LIN {X 0,Y 124.786,Z 596.16,A -85,B 0,C 180,E1 -33288.67,E2 -33288.67} C_VEL
LIN {X 0,Y 121.331,Z 587.817,A -85,B 0,C 180,E1 -33295.862,E2 -33295.862} C_VEL
LIN {X 0,Y 119.937,Z 579.475,A -85,B 0,C 180,E1 -33301.975,E2 -33301.975} C_VEL
LIN {X 0,Y 119.69,Z 571.877,A -85,B 0,C 180,E1 -33306.721,E2 -33306.721} C_VEL
LIN {X 0,Y 119.661,Z 563.812,A -85,B 0,C 180,E1 -33310.967,E2 -33310.967} C_VEL
LIN {X 0,Y 119.744,Z 553.937,A -85,B 0,C 180,E1 -33315.262,E2 -33315.262} C_VEL
LIN {X 0,Y 120.033,Z 541.878,A -85,B 0,C 180,E1 -33319.604,E2 -33319.604} C_VEL
LIN {X 0,Y 120.66,Z 528.353,A -85,B 0,C 180,E1 -33323.521,E2 -33323.521} C_VEL
LIN {X 0,Y 121.53,Z 514.293,A -85,B 0,C 180,E1 -33326.761,E2 -33326.761} C_VEL
LIN {X 0,Y 122.326,Z 501.194,A -85,B 0,C 180,E1 -33329.125,E2 -33329.125} C_VEL
LIN {X 0,Y 123.248,Z 486.148,A -85,B 0,C 180,E1 -33331.168,E2 -33331.168} C_VEL
LIN {X 0,Y 124.935,Z 446.734,A -85,B 0,C 180,E1 -33335.322,E2 -33335.322} C_VEL
LIN {X 0,Y 125.796,Z 425.42,A -85,B 0,C 180,E1 -33337.518,E2 -33337.518} C_VEL
LIN {X 0,Y 125.894,Z 429.15,A -85,B 0,C 180,E1 -33338,E2 -33338} C_VEL
LIN {X 0,Y 126.482,Z 430.582,A -85,B 0,C 180,E1 -33338.589,E2 -33338.589} C_VEL
LIN {X 0,Y 127.237,Z 430.409,A -85,B 0,C 180,E1 -33339.115,E2 -33339.115} C_VEL
LIN {X 0,Y 128.762,Z 427.949,A -85,B 0,C 180,E1 -33339.926,E2 -33339.926} C_VEL
LIN {X 0,Y 130.986,Z 422.371,A -85,B 0,C 180,E1 -33340.854,E2 -33340.854} C_VEL
LIN {X 0,Y 134.629,Z 410.741,A -85,B 0,C 180,E1 -33342.038,E2 -33342.038} C_VEL
LIN {X 0,Y 136.236,Z 405.229,A -85,B 0,C 180,E1 -33342.495,E2 -33342.495} C_VEL
LIN {X 0,Y 138.125,Z 404.048,A -85,B 0,C 180,E1 -33343.473,E2 -33343.473} C_VEL
LIN {X 0,Y 141.272,Z 399.719,A -85,B 0,C 180,E1 -33344.805,E2 -33344.805} C_VEL
LIN {X 0,Y 143.724,Z 394.588,A -85,B 0,C 180,E1 -33345.638,E2 -33345.638} C_VEL
LIN {X 0,Y 145.398,Z 390.211,A -85,B 0,C 180,E1 -33346.116,E2 -33346.116} C_VEL
LIN {X 0,Y 148.34,Z 387.317,A -85,B 0,C 180,E1 -33347.273,E2 -33347.273} C_VEL
LIN {X 0,Y 149.643,Z 385.499,A -85,B 0,C 180,E1 -33347.724,E2 -33347.724} C_VEL
LIN {X 0,Y 153.065,Z 391.957,A -85,B 0,C 180,E1 -33349.628,E2 -33349.628} C_VEL
LIN {X 0,Y 157.455,Z 401.657,A -85,B 0,C 180,E1 -33351.951,E2 -33351.951} C_VEL
LIN {X 0,Y 153.089,Z 461.487,A -85,B 0,C 180,E1 -33354.305,E2 -33354.305} C_VEL
LIN {X 0,Y 151.198,Z 475.824,A -85,B 0,C 180,E1 -33355.316,E2 -33355.316} C_VEL
LIN {X 0,Y 148.632,Z 489.602,A -85,B 0,C 180,E1 -33356.774,E2 -33356.774} C_VEL
LIN {X 0,Y 145.094,Z 503.399,A -85,B 0,C 180,E1 -33358.73,E2 -33358.73} C_VEL
LIN {X 0,Y 141.064,Z 515.819,A -85,B 0,C 180,E1 -33361.037,E2 -33361.037} C_VEL
LIN {X 0,Y 136.983,Z 527.133,A -85,B 0,C 180,E1 -33363.823,E2 -33363.823} C_VEL
LIN {X 0,Y 134.16,Z 534.593,A -85,B 0,C 180,E1 -33366.125,E2 -33366.125} C_VEL
LIN {X 0,Y 130.069,Z 543.848,A -85,B 0,C 180,E1 -33369.503,E2 -33369.503} C_VEL
LIN {X 0,Y 126.03,Z 553.071,A -85,B 0,C 180,E1 -33373.858,E2 -33373.858} C_VEL
LIN {X 0,Y 122.461,Z 560.792,A -85,B 0,C 180,E1 -33378.444,E2 -33378.444} C_VEL
LIN {X 0,Y 119.77,Z 567.796,A -85,B 0,C 180,E1 -33383.825,E2 -33383.825} C_VEL
LIN {X 0,Y 117.465,Z 574.032,A -85,B 0,C 180,E1 -33389.992,E2 -33389.992} C_VEL
LIN {X 0,Y 115.944,Z 579.238,A -85,B 0,C 180,E1 -33396.931,E2 -33396.931} C_VEL
LIN {X 0,Y 115.95,Z 582.927,A -85,B 0,C 180,E1 -33403.974,E2 -33403.974} C_VEL
LIN {X 0,Y 117.079,Z 585.235,A -85,B 0,C 180,E1 -33411.027,E2 -33411.027} C_VEL
LIN {X 0,Y 119.806,Z 586.166,A -85,B 0,C 180,E1 -33417.876,E2 -33417.876} C_VEL
LIN {X 0,Y 123.903,Z 585.74,A -85,B 0,C 180,E1 -33424.414,E2 -33424.414} C_VEL
LIN {X 0,Y 129.421,Z 583.919,A -85,B 0,C 180,E1 -33430.49,E2 -33430.49} C_VEL
LIN {X 0,Y 136.163,Z 580.628,A -85,B 0,C 180,E1 -33436.058,E2 -33436.058} C_VEL
LIN {X 0,Y 144.038,Z 575.777,A -85,B 0,C 180,E1 -33441.072,E2 -33441.072} C_VEL
LIN {X 0,Y 150.576,Z 571.039,A -85,B 0,C 180,E1 -33444.482,E2 -33444.482} C_VEL
LIN {X 0,Y 158.257,Z 564.569,A -85,B 0,C 180,E1 -33447.919,E2 -33447.919} C_VEL
LIN {X 0,Y 166.233,Z 556.792,A -85,B 0,C 180,E1 -33450.952,E2 -33450.952} C_VEL
LIN {X 0,Y 174.638,Z 547.262,A -85,B 0,C 180,E1 -33453.688,E2 -33453.688} C_VEL
LIN {X 0,Y 182.245,Z 537.131,A -85,B 0,C 180,E1 -33455.881,E2 -33455.881} C_VEL
LIN {X 0,Y 189.205,Z 526.13,A -85,B 0,C 180,E1 -33457.729,E2 -33457.729} C_VEL
LIN {X 0,Y 195.617,Z 514.012,A -85,B 0,C 180,E1 -33459.285,E2 -33459.285} C_VEL
LIN {X 0,Y 200.66,Z 502.302,A -85,B 0,C 180,E1 -33460.457,E2 -33460.457} C_VEL
LIN {X 0,Y 204.641,Z 490.765,A -85,B 0,C 180,E1 -33461.368,E2 -33461.368} C_VEL
LIN {X 0,Y 208.302,Z 476.926,A -85,B 0,C 180,E1 -33462.188,E2 -33462.188} C_VEL
LIN {X 0,Y 210.928,Z 462.395,A -85,B 0,C 180,E1 -33462.766,E2 -33462.766} C_VEL
LIN {X 0,Y 212.271,Z 449.436,A -85,B 0,C 180,E1 -33463.132,E2 -33463.132} C_VEL
LIN {X 0,Y 208.709,Z 441.693,A -85,B 0,C 180,E1 -33466.336,E2 -33466.336} C_VEL
LIN {X 0,Y 205.63,Z 435.551,A -85,B 0,C 180,E1 -33469.652,E2 -33469.652} C_VEL
LIN {X 0,Y 204.019,Z 432.479,A -85,B 0,C 180,E1 -33471.734,E2 -33471.734} C_VEL
LIN {X 0,Y 202.594,Z 429.652,A -85,B 0,C 180,E1 -33473.922,E2 -33473.922} C_VEL
LIN {X 0,Y 200.884,Z 426.052,A -85,B 0,C 180,E1 -33477.361,E2 -33477.361} C_VEL
LIN {X 0,Y 199.415,Z 422.655,A -85,B 0,C 180,E1 -33482.791,E2 -33482.791} C_VEL
LIN {X 0,Y 199.313,Z 422.048,A -85,B 0,C 180,E1 -33484.03,E2 -33484.03} C_VEL
LIN {X 0,Y 199.267,Z 422.448,A -85,B 0,C 180,E1 -33487.194,E2 -33487.194} C_VEL
LIN {X 0,Y 199.912,Z 425.362,A -85,B 0,C 180,E1 -33491.492,E2 -33491.492} C_VEL
LIN {X 0,Y 201.079,Z 428.272,A -85,B 0,C 180,E1 -33494.757,E2 -33494.757} C_VEL
LIN {X 0,Y 202.993,Z 433.534,A -85,B 0,C 180,E1 -33498.477,E2 -33498.477} C_VEL
LIN {X 0,Y 204.769,Z 438.369,A -85,B 0,C 180,E1 -33501.117,E2 -33501.117} C_VEL
LIN {X 0,Y 206.448,Z 442.889,A -85,B 0,C 180,E1 -33503.209,E2 -33503.209} C_VEL
LIN {X 0,Y 209.032,Z 450.588,A -85,B 0,C 180,E1 -33506.025,E2 -33506.025} C_VEL
LIN {X 0,Y 211.441,Z 458.554,A -85,B 0,C 180,E1 -33508.37,E2 -33508.37} C_VEL
LIN {X 0,Y 209.275,Z 476.668,A -85,B 0,C 180,E1 -33508.865,E2 -33508.865} C_VEL
LIN {X 0,Y 206.148,Z 491.123,A -85,B 0,C 180,E1 -33509.399,E2 -33509.399} C_VEL
LIN {X 0,Y 201.995,Z 504.823,A -85,B 0,C 180,E1 -33510.158,E2 -33510.158} C_VEL
LIN {X 0,Y 196.356,Z 518.574,A -85,B 0,C 180,E1 -33511.126,E2 -33511.126} C_VEL
LIN {X 0,Y 189.751,Z 531.543,A -85,B 0,C 180,E1 -33512.403,E2 -33512.403} C_VEL
LIN {X 0,Y 182.631,Z 543.22,A -85,B 0,C 180,E1 -33513.976,E2 -33513.976} C_VEL
LIN {X 0,Y 174.977,Z 553.813,A -85,B 0,C 180,E1 -33515.854,E2 -33515.854} C_VEL
LIN {X 0,Y 167.023,Z 563.393,A -85,B 0,C 180,E1 -33518.168,E2 -33518.168} C_VEL
LIN {X 0,Y 158.164,Z 572.605,A -85,B 0,C 180,E1 -33521.172,E2 -33521.172} C_VEL
LIN {X 0,Y 149.131,Z 580.565,A -85,B 0,C 180,E1 -33524.792,E2 -33524.792} C_VEL
LIN {X 0,Y 142.073,Z 586.074,A -85,B 0,C 180,E1 -33528.284,E2 -33528.284} C_VEL
LIN {X 0,Y 134.207,Z 591.389,A -85,B 0,C 180,E1 -33533.126,E2 -33533.126} C_VEL
LIN {X 0,Y 129.096,Z 594.407,A -85,B 0,C 180,E1 -33537.15,E2 -33537.15} C_VEL
LIN {X 0,Y 123.515,Z 597.242,A -85,B 0,C 180,E1 -33543.03,E2 -33543.03} C_VEL
LIN {X 0,Y 119.322,Z 598.763,A -85,B 0,C 180,E1 -33549.386,E2 -33549.386} C_VEL
LIN {X 0,Y 116.711,Z 599.003,A -85,B 0,C 180,E1 -33556.119,E2 -33556.119} C_VEL
LIN {X 0,Y 115.778,Z 597.964,A -85,B 0,C 180,E1 -33563.059,E2 -33563.059} C_VEL
LIN {X 0,Y 116.649,Z 595.626,A -85,B 0,C 180,E1 -33570.008,E2 -33570.008} C_VEL
LIN {X 0,Y 117.97,Z 592.905,A -85,B 0,C 180,E1 -33575.118,E2 -33575.118} C_VEL
LIN {X 0,Y 120.631,Z 587.981,A -85,B 0,C 180,E1 -33581.734,E2 -33581.734} C_VEL
LIN {X 0,Y 121.219,Z 587.202,A -85,B 0,C 180,E1 -33582.735,E2 -33582.735} C_VEL
LIN {X 0,Y 122.769,Z 595.357,A -85,B 0,C 180,E1 -33590.027,E2 -33590.027} C_VEL
LIN {X 0,Y 126.327,Z 601.493,A -85,B 0,C 180,E1 -33596.34,E2 -33596.34} C_VEL
LIN {X 0,Y 131.608,Z 606.467,A -85,B 0,C 180,E1 -33602.164,E2 -33602.164} C_VEL
LIN {X 0,Y 138.447,Z 610.396,A -85,B 0,C 180,E1 -33607.389,E2 -33607.389} C_VEL
LIN {X 0,Y 146.713,Z 613.364,A -85,B 0,C 180,E1 -33611.951,E2 -33611.951} C_VEL
LIN {X 0,Y 156.108,Z 615.34,A -85,B 0,C 180,E1 -33615.89,E2 -33615.89} C_VEL
LIN {X 0,Y 160.999,Z 615.939,A -85,B 0,C 180,E1 -33617.706,E2 -33617.706} C_VEL
LIN {X 0,Y 174.126,Z 616.495,A -85,B 0,C 180,E1 -33621.419,E2 -33621.419} C_VEL
LIN {X 0,Y 173.938,Z 616.434,A -85,B 0,C 180,E1 -33622.116,E2 -33622.116} C_VEL
LIN {X 0,Y 160.784,Z 615.271,A -85,B 0,C 180,E1 -33625.875,E2 -33625.875} C_VEL
LIN {X 0,Y 156.765,Z 614.568,A -85,B 0,C 180,E1 -33627.278,E2 -33627.278} C_VEL
LIN {X 0,Y 152.254,Z 613.642,A -85,B 0,C 180,E1 -33628.646,E2 -33628.646} C_VEL
LIN {X 0,Y 143.994,Z 611.406,A -85,B 0,C 180,E1 -33630.571,E2 -33630.571} C_VEL
LIN {X 0,Y 136.123,Z 608.585,A -85,B 0,C 180,E1 -33632.734,E2 -33632.734} C_VEL
LIN {X 0,Y 132.323,Z 606.728,A -85,B 0,C 180,E1 -33634.498,E2 -33634.498} C_VEL
LIN {X 0,Y 124.716,Z 601.289,A -85,B 0,C 180,E1 -33640.307,E2 -33640.307} C_VEL
LIN {X 0,Y 119.272,Z 595.033,A -85,B 0,C 180,E1 -33646.414,E2 -33646.414} C_VEL
LIN {X 0,Y 115.309,Z 586.537,A -85,B 0,C 180,E1 -33653.898,E2 -33653.898} C_VEL
LIN {X 0,Y 113.702,Z 578.514,A -85,B 0,C 180,E1 -33660,E2 -33660} C_VEL
LIN {X 0,Y 113.254,Z 570.221,A -85,B 0,C 180,E1 -33665.428,E2 -33665.428} C_VEL
LIN {X 0,Y 113.172,Z 562.224,A -85,B 0,C 180,E1 -33669.799,E2 -33669.799} C_VEL
LIN {X 0,Y 113.119,Z 552.221,A -85,B 0,C 180,E1 -33674.34,E2 -33674.34} C_VEL
LIN {X 0,Y 113.329,Z 540.159,A -85,B 0,C 180,E1 -33678.825,E2 -33678.825} C_VEL
LIN {X 0,Y 113.895,Z 526.412,A -85,B 0,C 180,E1 -33682.963,E2 -33682.963} C_VEL
LIN {X 0,Y 114.665,Z 512.54,A -85,B 0,C 180,E1 -33686.287,E2 -33686.287} C_VEL
LIN {X 0,Y 115.445,Z 499.01,A -85,B 0,C 180,E1 -33688.79,E2 -33688.79} C_VEL
LIN {X 0,Y 116.398,Z 483.579,A -85,B 0,C 180,E1 -33690.904,E2 -33690.904} C_VEL
LIN {X 0,Y 117.412,Z 455.66,A -85,B 0,C 180,E1 -33694.069,E2 -33694.069} C_VEL
LIN {X 0,Y 117.335,Z 459.549,A -85,B 0,C 180,E1 -33694.547,E2 -33694.547} C_VEL
LIN {X 0,Y 117.688,Z 460.919,A -85,B 0,C 180,E1 -33695.078,E2 -33695.078} C_VEL
LIN {X 0,Y 118.411,Z 461.078,A -85,B 0,C 180,E1 -33695.742,E2 -33695.742} C_VEL
LIN {X 0,Y 119.571,Z 459.529,A -85,B 0,C 180,E1 -33696.509,E2 -33696.509} C_VEL
LIN {X 0,Y 121.511,Z 455.002,A -85,B 0,C 180,E1 -33697.508,E2 -33697.508} C_VEL
LIN {X 0,Y 125.038,Z 443.841,A -85,B 0,C 180,E1 -33698.949,E2 -33698.949} C_VEL
LIN {X 0,Y 126.718,Z 437.654,A -85,B 0,C 180,E1 -33699.502,E2 -33699.502} C_VEL
LIN {X 0,Y 128.858,Z 436.184,A -85,B 0,C 180,E1 -33700.814,E2 -33700.814} C_VEL
LIN {X 0,Y 131.063,Z 433.055,A -85,B 0,C 180,E1 -33701.927,E2 -33701.927} C_VEL
LIN {X 0,Y 133.524,Z 427.64,A -85,B 0,C 180,E1 -33702.918,E2 -33702.918} C_VEL
LIN {X 0,Y 137.067,Z 417.356,A -85,B 0,C 180,E1 -33704.031,E2 -33704.031} C_VEL
LIN {X 0,Y 139.189,Z 410.568,A -85,B 0,C 180,E1 -33704.606,E2 -33704.606} C_VEL
LIN {X 0,Y 141.994,Z 407.51,A -85,B 0,C 180,E1 -33705.802,E2 -33705.802} C_VEL
LIN {X 0,Y 145.407,Z 402.221,A -85,B 0,C 180,E1 -33707.039,E2 -33707.039} C_VEL
LIN {X 0,Y 148.252,Z 395.708,A -85,B 0,C 180,E1 -33707.851,E2 -33707.851} C_VEL
LIN {X 0,Y 148.691,Z 395.792,A -85,B 0,C 180,E1 -33708.051,E2 -33708.051} C_VEL
LIN {X 0,Y 152.379,Z 404.131,A -85,B 0,C 180,E1 -33710.183,E2 -33710.183} C_VEL
LIN {X 0,Y 147.971,Z 461.483,A -85,B 0,C 180,E1 -33712.442,E2 -33712.442} C_VEL
LIN {X 0,Y 145.99,Z 475.961,A -85,B 0,C 180,E1 -33713.463,E2 -33713.463} C_VEL
LIN {X 0,Y 143.317,Z 489.803,A -85,B 0,C 180,E1 -33714.944,E2 -33714.944} C_VEL
LIN {X 0,Y 139.617,Z 503.647,A -85,B 0,C 180,E1 -33716.927,E2 -33716.927} C_VEL
LIN {X 0,Y 135.409,Z 516.098,A -85,B 0,C 180,E1 -33719.274,E2 -33719.274} C_VEL
LIN {X 0,Y 131.124,Z 527.436,A -85,B 0,C 180,E1 -33722.126,E2 -33722.126} C_VEL
LIN {X 0,Y 127.655,Z 535.899,A -85,B 0,C 180,E1 -33724.826,E2 -33724.826} C_VEL
LIN {X 0,Y 122.703,Z 546.621,A -85,B 0,C 180,E1 -33729.089,E2 -33729.089} C_VEL
LIN {X 0,Y 118.483,Z 555.466,A -85,B 0,C 180,E1 -33733.683,E2 -33733.683} C_VEL
LIN {X 0,Y 115.065,Z 562.819,A -85,B 0,C 180,E1 -33738.581,E2 -33738.581} C_VEL
LIN {X 0,Y 112.169,Z 569.849,A -85,B 0,C 180,E1 -33744.617,E2 -33744.617} C_VEL
LIN {X 0,Y 110.295,Z 574.774,A -85,B 0,C 180,E1 -33749.991,E2 -33749.991} C_VEL
LIN {X 0,Y 108.824,Z 579.899,A -85,B 0,C 180,E1 -33757.387,E2 -33757.387} C_VEL
LIN {X 0,Y 108.933,Z 583.516,A -85,B 0,C 180,E1 -33764.895,E2 -33764.895} C_VEL
LIN {X 0,Y 110.333,Z 585.751,A -85,B 0,C 180,E1 -33772.38,E2 -33772.38} C_VEL
LIN {X 0,Y 113.426,Z 586.609,A -85,B 0,C 180,E1 -33779.595,E2 -33779.595} C_VEL
LIN {X 0,Y 117.947,Z 586.098,A -85,B 0,C 180,E1 -33786.421,E2 -33786.421} C_VEL
LIN {X 0,Y 124.017,Z 584.145,A -85,B 0,C 180,E1 -33792.757,E2 -33792.757} C_VEL
LIN {X 0,Y 131.181,Z 580.805,A -85,B 0,C 180,E1 -33798.365,E2 -33798.365} C_VEL
LIN {X 0,Y 139.548,Z 575.871,A -85,B 0,C 180,E1 -33803.414,E2 -33803.414} C_VEL
LIN {X 0,Y 146.442,Z 571.043,A -85,B 0,C 180,E1 -33806.815,E2 -33806.815} C_VEL
LIN {X 0,Y 155.021,Z 564.006,A -85,B 0,C 180,E1 -33810.419,E2 -33810.419} C_VEL
LIN {X 0,Y 164.143,Z 555.214,A -85,B 0,C 180,E1 -33813.638,E2 -33813.638} C_VEL
LIN {X 0,Y 172.976,Z 545.207,A -85,B 0,C 180,E1 -33816.28,E2 -33816.28} C_VEL
LIN {X 0,Y 180.814,Z 534.594,A -85,B 0,C 180,E1 -33818.374,E2 -33818.374} C_VEL
LIN {X 0,Y 187.404,Z 524.016,A -85,B 0,C 180,E1 -33819.998,E2 -33819.998} C_VEL
LIN {X 0,Y 193.906,Z 511.462,A -85,B 0,C 180,E1 -33821.463,E2 -33821.463} C_VEL
LIN {X 0,Y 199.431,Z 497.964,A -85,B 0,C 180,E1 -33822.704,E2 -33822.704} C_VEL
LIN {X 0,Y 203.545,Z 485.099,A -85,B 0,C 180,E1 -33823.565,E2 -33823.565} C_VEL
LIN {X 0,Y 206.723,Z 471.452,A -85,B 0,C 180,E1 -33824.244,E2 -33824.244} C_VEL
LIN {X 0,Y 208.917,Z 456.849,A -85,B 0,C 180,E1 -33824.703,E2 -33824.703} C_VEL
LIN {X 0,Y 209.235,Z 453.245,A -85,B 0,C 180,E1 -33824.827,E2 -33824.827} C_VEL
LIN {X 0,Y 206.029,Z 446.048,A -85,B 0,C 180,E1 -33828.043,E2 -33828.043} C_VEL
LIN {X 0,Y 203.28,Z 440.227,A -85,B 0,C 180,E1 -33831.454,E2 -33831.454} C_VEL
LIN {X 0,Y 201.253,Z 436.234,A -85,B 0,C 180,E1 -33834.633,E2 -33834.633} C_VEL
LIN {X 0,Y 199.726,Z 432.805,A -85,B 0,C 180,E1 -33837.99,E2 -33837.99} C_VEL
LIN {X 0,Y 198.487,Z 429.491,A -85,B 0,C 180,E1 -33843.274,E2 -33843.274} C_VEL
LIN {X 0,Y 198.439,Z 429.08,A -85,B 0,C 180,E1 -33844.048,E2 -33844.048} C_VEL
LIN {X 0,Y 198.374,Z 429.388,A -85,B 0,C 180,E1 -33846.844,E2 -33846.844} C_VEL
LIN {X 0,Y 198.914,Z 432.268,A -85,B 0,C 180,E1 -33851.103,E2 -33851.103} C_VEL
LIN {X 0,Y 199.921,Z 435.026,A -85,B 0,C 180,E1 -33854.197,E2 -33854.197} C_VEL
LIN {X 0,Y 201.65,Z 440.167,A -85,B 0,C 180,E1 -33857.847,E2 -33857.847} C_VEL
LIN {X 0,Y 203.342,Z 445.121,A -85,B 0,C 180,E1 -33860.544,E2 -33860.544} C_VEL
LIN {X 0,Y 205.161,Z 450.553,A -85,B 0,C 180,E1 -33862.959,E2 -33862.959} C_VEL
LIN {X 0,Y 207.594,Z 458.577,A -85,B 0,C 180,E1 -33865.748,E2 -33865.748} C_VEL
LIN {X 0,Y 208.434,Z 461.626,A -85,B 0,C 180,E1 -33866.642,E2 -33866.642} C_VEL
LIN {X 0,Y 206.397,Z 477.2,A -85,B 0,C 180,E1 -33867.067,E2 -33867.067} C_VEL
LIN {X 0,Y 203.377,Z 490.75,A -85,B 0,C 180,E1 -33867.569,E2 -33867.569} C_VEL
LIN {X 0,Y 199.473,Z 503.426,A -85,B 0,C 180,E1 -33868.234,E2 -33868.234} C_VEL
LIN {X 0,Y 194.323,Z 516.192,A -85,B 0,C 180,E1 -33869.073,E2 -33869.073} C_VEL
LIN {X 0,Y 188.264,Z 528.261,A -85,B 0,C 180,E1 -33870.126,E2 -33870.126} C_VEL
LIN {X 0,Y 180.973,Z 540.45,A -85,B 0,C 180,E1 -33871.637,E2 -33871.637} C_VEL
LIN {X 0,Y 173.778,Z 550.545,A -85,B 0,C 180,E1 -33873.253,E2 -33873.253} C_VEL
LIN {X 0,Y 165.433,Z 560.598,A -85,B 0,C 180,E1 -33875.42,E2 -33875.42} C_VEL
LIN {X 0,Y 157.449,Z 568.979,A -85,B 0,C 180,E1 -33877.859,E2 -33877.859} C_VEL
LIN {X 0,Y 148.528,Z 577.025,A -85,B 0,C 180,E1 -33881.025,E2 -33881.025} C_VEL
LIN {X 0,Y 141.32,Z 582.732,A -85,B 0,C 180,E1 -33884.07,E2 -33884.07} C_VEL
LIN {X 0,Y 132.55,Z 588.754,A -85,B 0,C 180,E1 -33888.669,E2 -33888.669} C_VEL
LIN {X 0,Y 126.69,Z 592.272,A -85,B 0,C 180,E1 -33892.553,E2 -33892.553} C_VEL
LIN {X 0,Y 120.043,Z 595.721,A -85,B 0,C 180,E1 -33898.332,E2 -33898.332} C_VEL
LIN {X 0,Y 114.767,Z 597.826,A -85,B 0,C 180,E1 -33904.718,E2 -33904.718} C_VEL
LIN {X 0,Y 111.035,Z 598.638,A -85,B 0,C 180,E1 -33911.624,E2 -33911.624} C_VEL
LIN {X 0,Y 109.07,Z 598.173,A -85,B 0,C 180,E1 -33918.901,E2 -33918.901} C_VEL
LIN {X 0,Y 108.951,Z 596.419,A -85,B 0,C 180,E1 -33926.323,E2 -33926.323} C_VEL
LIN {X 0,Y 110.422,Z 593.303,A -85,B 0,C 180,E1 -33933.646,E2 -33933.646} C_VEL
LIN {X 0,Y 112.818,Z 588.667,A -85,B 0,C 180,E1 -33940.743,E2 -33940.743} C_VEL
LIN {X 0,Y 114.987,Z 585.569,A -85,B 0,C 180,E1 -33944.562,E2 -33944.562} C_VEL
LIN {X 0,Y 116.57,Z 592.795,A -85,B 0,C 180,E1 -33951.141,E2 -33951.141} C_VEL
LIN {X 0,Y 120.323,Z 599.273,A -85,B 0,C 180,E1 -33957.765,E2 -33957.765} C_VEL
LIN {X 0,Y 125.881,Z 604.571,A -85,B 0,C 180,E1 -33963.818,E2 -33963.818} C_VEL
LIN {X 0,Y 133.025,Z 608.814,A -85,B 0,C 180,E1 -33969.196,E2 -33969.196} C_VEL
LIN {X 0,Y 141.607,Z 612.103,A -85,B 0,C 180,E1 -33973.837,E2 -33973.837} C_VEL
LIN {X 0,Y 151.3,Z 614.449,A -85,B 0,C 180,E1 -33977.801,E2 -33977.801} C_VEL
LIN {X 0,Y 156.332,Z 615.243,A -85,B 0,C 180,E1 -33979.621,E2 -33979.621} C_VEL
LIN {X 0,Y 161.752,Z 615.823,A -85,B 0,C 180,E1 -33981.22,E2 -33981.22} C_VEL
LIN {X 0,Y 162.342,Z 615.821,A -85,B 0,C 180,E1 -33982.117,E2 -33982.117} C_VEL
LIN {X 0,Y 150.236,Z 613.619,A -85,B 0,C 180,E1 -33985.98,E2 -33985.98} C_VEL
LIN {X 0,Y 140.388,Z 610.55,A -85,B 0,C 180,E1 -33990.07,E2 -33990.07} C_VEL
LIN {X 0,Y 132.323,Z 606.728,A -85,B 0,C 180,E1 -33994.498,E2 -33994.498} C_VEL
LIN {X 0,Y 128.761,Z 604.724,A -85,B 0,C 180,E1 -33996.373,E2 -33996.373} C_VEL
LIN {X 0,Y 122.107,Z 600.646,A -85,B 0,C 180,E1 -33999.171,E2 -33999.171} C_VEL
LIN {X 0,Y 116.06,Z 596.039,A -85,B 0,C 180,E1 -34002.235,E2 -34002.235} C_VEL
LIN {X 0,Y 113.558,Z 593.239,A -85,B 0,C 180,E1 -34004.511,E2 -34004.511} C_VEL
LIN {X 0,Y 109.164,Z 584.071,A -85,B 0,C 180,E1 -34012.627,E2 -34012.627} C_VEL
LIN {X 0,Y 107.266,Z 574.43,A -85,B 0,C 180,E1 -34020,E2 -34020} C_VEL
LIN {X 0,Y 106.866,Z 565.85,A -85,B 0,C 180,E1 -34025.542,E2 -34025.542} C_VEL
LIN {X 0,Y 106.664,Z 557.826,A -85,B 0,C 180,E1 -34029.879,E2 -34029.879} C_VEL
LIN {X 0,Y 106.55,Z 546.82,A -85,B 0,C 180,E1 -34034.758,E2 -34034.758} C_VEL
LIN {X 0,Y 106.722,Z 534.753,A -85,B 0,C 180,E1 -34039.157,E2 -34039.157} C_VEL
LIN {X 0,Y 107.282,Z 521.62,A -85,B 0,C 180,E1 -34043.063,E2 -34043.063} C_VEL
LIN {X 0,Y 108.106,Z 507.145,A -85,B 0,C 180,E1 -34046.451,E2 -34046.451} C_VEL
LIN {X 0,Y 109.001,Z 491.242,A -85,B 0,C 180,E1 -34049.208,E2 -34049.208} C_VEL
LIN {X 0,Y 109.682,Z 478.193,A -85,B 0,C 180,E1 -34050.915,E2 -34050.915} C_VEL
LIN {X 0,Y 109.496,Z 480.871,A -85,B 0,C 180,E1 -34051.684,E2 -34051.684} C_VEL
LIN {X 0,Y 109.763,Z 481.597,A -85,B 0,C 180,E1 -34052.246,E2 -34052.246} C_VEL
LIN {X 0,Y 110.477,Z 481.669,A -85,B 0,C 180,E1 -34053.05,E2 -34053.05} C_VEL
LIN {X 0,Y 112.022,Z 479.943,A -85,B 0,C 180,E1 -34054.075,E2 -34054.075} C_VEL
LIN {X 0,Y 114.326,Z 475.997,A -85,B 0,C 180,E1 -34055.144,E2 -34055.144} C_VEL
LIN {X 0,Y 117.293,Z 468.83,A -85,B 0,C 180,E1 -34056.136,E2 -34056.136} C_VEL
LIN {X 0,Y 117.633,Z 468.038,A -85,B 0,C 180,E1 -34056.279,E2 -34056.279} C_VEL
LIN {X 0,Y 119.451,Z 467.02,A -85,B 0,C 180,E1 -34057.604,E2 -34057.604} C_VEL
LIN {X 0,Y 121.585,Z 464.328,A -85,B 0,C 180,E1 -34058.793,E2 -34058.793} C_VEL
LIN {X 0,Y 124.09,Z 459.25,A -85,B 0,C 180,E1 -34059.947,E2 -34059.947} C_VEL
LIN {X 0,Y 127.515,Z 449.401,A -85,B 0,C 180,E1 -34061.236,E2 -34061.236} C_VEL
LIN {X 0,Y 129.497,Z 442.974,A -85,B 0,C 180,E1 -34061.887,E2 -34061.887} C_VEL
LIN {X 0,Y 132.513,Z 439.608,A -85,B 0,C 180,E1 -34063.406,E2 -34063.406} C_VEL
LIN {X 0,Y 135.451,Z 434.484,A -85,B 0,C 180,E1 -34064.615,E2 -34064.615} C_VEL
LIN {X 0,Y 139.264,Z 424.911,A -85,B 0,C 180,E1 -34065.826,E2 -34065.826} C_VEL
LIN {X 0,Y 142.557,Z 415.067,A -85,B 0,C 180,E1 -34066.675,E2 -34066.675} C_VEL
LIN {X 0,Y 146.69,Z 409.773,A -85,B 0,C 180,E1 -34068.187,E2 -34068.187} C_VEL
LIN {X 0,Y 147.128,Z 409.134,A -85,B 0,C 180,E1 -34068.334,E2 -34068.334} C_VEL
LIN {X 0,Y 142.895,Z 462.6,A -85,B 0,C 180,E1 -34070.52,E2 -34070.52} C_VEL
LIN {X 0,Y 140.817,Z 476.847,A -85,B 0,C 180,E1 -34071.546,E2 -34071.546} C_VEL
LIN {X 0,Y 137.852,Z 491.138,A -85,B 0,C 180,E1 -34073.107,E2 -34073.107} C_VEL
LIN {X 0,Y 134.287,Z 503.896,A -85,B 0,C 180,E1 -34074.979,E2 -34074.979} C_VEL
LIN {X 0,Y 129.878,Z 516.382,A -85,B 0,C 180,E1 -34077.355,E2 -34077.355} C_VEL
LIN {X 0,Y 125.392,Z 527.738,A -85,B 0,C 180,E1 -34080.272,E2 -34080.272} C_VEL
LIN {X 0,Y 122.218,Z 535.239,A -85,B 0,C 180,E1 -34082.702,E2 -34082.702} C_VEL
LIN {X 0,Y 116.891,Z 546.146,A -85,B 0,C 180,E1 -34087.068,E2 -34087.068} C_VEL
LIN {X 0,Y 112.387,Z 555.135,A -85,B 0,C 180,E1 -34091.834,E2 -34091.834} C_VEL
LIN {X 0,Y 108.629,Z 562.624,A -85,B 0,C 180,E1 -34096.948,E2 -34096.948} C_VEL
LIN {X 0,Y 105.883,Z 568.856,A -85,B 0,C 180,E1 -34102.388,E2 -34102.388} C_VEL
LIN {X 0,Y 103.708,Z 574.027,A -85,B 0,C 180,E1 -34108.055,E2 -34108.055} C_VEL
LIN {X 0,Y 102.197,Z 578.235,A -85,B 0,C 180,E1 -34113.92,E2 -34113.92} C_VEL
LIN {X 0,Y 101.607,Z 582.514,A -85,B 0,C 180,E1 -34121.925,E2 -34121.925} C_VEL
LIN {X 0,Y 101.943,Z 584.107,A -85,B 0,C 180,E1 -34125.942,E2 -34125.942} C_VEL
LIN {X 0,Y 103.625,Z 586.269,A -85,B 0,C 180,E1 -34133.916,E2 -34133.916} C_VEL
LIN {X 0,Y 107.135,Z 587.04,A -85,B 0,C 180,E1 -34141.525,E2 -34141.525} C_VEL
LIN {X 0,Y 112.129,Z 586.435,A -85,B 0,C 180,E1 -34148.647,E2 -34148.647} C_VEL
LIN {X 0,Y 118.658,Z 584.434,A -85,B 0,C 180,E1 -34155.09,E2 -34155.09} C_VEL
LIN {X 0,Y 126.428,Z 580.983,A -85,B 0,C 180,E1 -34160.849,E2 -34160.849} C_VEL
LIN {X 0,Y 135.309,Z 575.965,A -85,B 0,C 180,E1 -34165.906,E2 -34165.906} C_VEL
LIN {X 0,Y 142.563,Z 571.046,A -85,B 0,C 180,E1 -34169.281,E2 -34169.281} C_VEL
LIN {X 0,Y 151.551,Z 563.911,A -85,B 0,C 180,E1 -34172.82,E2 -34172.82} C_VEL
LIN {X 0,Y 159.646,Z 556.379,A -85,B 0,C 180,E1 -34175.544,E2 -34175.544} C_VEL
LIN {X 0,Y 168.161,Z 547.206,A -85,B 0,C 180,E1 -34177.983,E2 -34177.983} C_VEL
LIN {X 0,Y 176.786,Z 536.162,A -85,B 0,C 180,E1 -34180.201,E2 -34180.201} C_VEL
LIN {X 0,Y 184.17,Z 524.753,A -85,B 0,C 180,E1 -34181.935,E2 -34181.935} C_VEL
LIN {X 0,Y 190.198,Z 513.639,A -85,B 0,C 180,E1 -34183.215,E2 -34183.215} C_VEL
LIN {X 0,Y 195.872,Z 500.616,A -85,B 0,C 180,E1 -34184.406,E2 -34184.406} C_VEL
LIN {X 0,Y 200.195,Z 487.982,A -85,B 0,C 180,E1 -34185.281,E2 -34185.281} C_VEL
LIN {X 0,Y 203.716,Z 473.937,A -85,B 0,C 180,E1 -34186.01,E2 -34186.01} C_VEL
LIN {X 0,Y 206.04,Z 460.105,A -85,B 0,C 180,E1 -34186.461,E2 -34186.461} C_VEL
LIN {X 0,Y 206.362,Z 457.174,A -85,B 0,C 180,E1 -34186.568,E2 -34186.568} C_VEL
LIN {X 0,Y 203.461,Z 450.404,A -85,B 0,C 180,E1 -34189.9,E2 -34189.9} C_VEL
LIN {X 0,Y 201.427,Z 445.977,A -85,B 0,C 180,E1 -34192.758,E2 -34192.758} C_VEL
LIN {X 0,Y 200.008,Z 442.93,A -85,B 0,C 180,E1 -34195.229,E2 -34195.229} C_VEL
LIN {X 0,Y 198.692,Z 439.705,A -85,B 0,C 180,E1 -34198.359,E2 -34198.359} C_VEL
LIN {X 0,Y 197.564,Z 436.124,A -85,B 0,C 180,E1 -34204.066,E2 -34204.066} C_VEL
LIN {X 0,Y 197.485,Z 436.52,A -85,B 0,C 180,E1 -34206.78,E2 -34206.78} C_VEL
LIN {X 0,Y 197.951,Z 439.285,A -85,B 0,C 180,E1 -34210.835,E2 -34210.835} C_VEL
LIN {X 0,Y 198.825,Z 441.948,A -85,B 0,C 180,E1 -34213.757,E2 -34213.757} C_VEL
LIN {X 0,Y 200.246,Z 446.5,A -85,B 0,C 180,E1 -34217.035,E2 -34217.035} C_VEL
LIN {X 0,Y 201.672,Z 451.064,A -85,B 0,C 180,E1 -34219.553,E2 -34219.553} C_VEL
LIN {X 0,Y 203.369,Z 456.653,A -85,B 0,C 180,E1 -34222.049,E2 -34222.049} C_VEL
LIN {X 0,Y 205.56,Z 464.532,A -85,B 0,C 180,E1 -34224.8,E2 -34224.8} C_VEL
LIN {X 0,Y 205.315,Z 467.567,A -85,B 0,C 180,E1 -34224.973,E2 -34224.973} C_VEL
LIN {X 0,Y 202.838,Z 482.067,A -85,B 0,C 180,E1 -34225.38,E2 -34225.38} C_VEL
LIN {X 0,Y 199.197,Z 495.849,A -85,B 0,C 180,E1 -34225.925,E2 -34225.925} C_VEL
LIN {X 0,Y 194.117,Z 510.107,A -85,B 0,C 180,E1 -34226.751,E2 -34226.751} C_VEL
LIN {X 0,Y 187.901,Z 523.29,A -85,B 0,C 180,E1 -34227.72,E2 -34227.72} C_VEL
LIN {X 0,Y 181.052,Z 535.191,A -85,B 0,C 180,E1 -34228.932,E2 -34228.932} C_VEL
LIN {X 0,Y 172.92,Z 547.045,A -85,B 0,C 180,E1 -34230.609,E2 -34230.609} C_VEL
LIN {X 0,Y 164.213,Z 557.661,A -85,B 0,C 180,E1 -34232.615,E2 -34232.615} C_VEL
LIN {X 0,Y 155.906,Z 566.448,A -85,B 0,C 180,E1 -34234.935,E2 -34234.935} C_VEL
LIN {X 0,Y 146.563,Z 574.914,A -85,B 0,C 180,E1 -34237.961,E2 -34237.961} C_VEL
LIN {X 0,Y 137.612,Z 581.831,A -85,B 0,C 180,E1 -34241.43,E2 -34241.43} C_VEL
LIN {X 0,Y 129.521,Z 587.253,A -85,B 0,C 180,E1 -34245.341,E2 -34245.341} C_VEL
LIN {X 0,Y 121.116,Z 592.068,A -85,B 0,C 180,E1 -34250.506,E2 -34250.506} C_VEL
LIN {X 0,Y 114.032,Z 595.439,A -85,B 0,C 180,E1 -34256.45,E2 -34256.45} C_VEL
LIN {X 0,Y 108.372,Z 597.471,A -85,B 0,C 180,E1 -34263.111,E2 -34263.111} C_VEL
LIN {X 0,Y 104.289,Z 598.213,A -85,B 0,C 180,E1 -34270.388,E2 -34270.388} C_VEL
LIN {X 0,Y 102.103,Z 597.682,A -85,B 0,C 180,E1 -34278.133,E2 -34278.133} C_VEL
LIN {X 0,Y 101.858,Z 595.86,A -85,B 0,C 180,E1 -34286.067,E2 -34286.067} C_VEL
LIN {X 0,Y 103.358,Z 592.68,A -85,B 0,C 180,E1 -34293.895,E2 -34293.895} C_VEL
LIN {X 0,Y 105.9,Z 587.976,A -85,B 0,C 180,E1 -34301.454,E2 -34301.454} C_VEL
LIN {X 0,Y 108.931,Z 583.824,A -85,B 0,C 180,E1 -34306.588,E2 -34306.588} C_VEL
LIN {X 0,Y 111.325,Z 591.878,A -85,B 0,C 180,E1 -34314.149,E2 -34314.149} C_VEL
LIN {X 0,Y 115.801,Z 598.387,A -85,B 0,C 180,E1 -34320.949,E2 -34320.949} C_VEL
LIN {X 0,Y 122.05,Z 603.738,A -85,B 0,C 180,E1 -34327.065,E2 -34327.065} C_VEL
LIN {X 0,Y 127.776,Z 607.095,A -85,B 0,C 180,E1 -34331.143,E2 -34331.143} C_VEL
LIN {X 0,Y 136.682,Z 610.701,A -85,B 0,C 180,E1 -34335.853,E2 -34335.853} C_VEL
LIN {X 0,Y 146.676,Z 613.374,A -85,B 0,C 180,E1 -34339.834,E2 -34339.834} C_VEL
LIN {X 0,Y 151.88,Z 614.346,A -85,B 0,C 180,E1 -34341.639,E2 -34341.639} C_VEL
LIN {X 0,Y 149.701,Z 613.874,A -85,B 0,C 180,E1 -34342.536,E2 -34342.536} C_VEL
LIN {X 0,Y 139.154,Z 610.834,A -85,B 0,C 180,E1 -34346.379,E2 -34346.379} C_VEL
LIN {X 0,Y 127.585,Z 605.595,A -85,B 0,C 180,E1 -34352.183,E2 -34352.183} C_VEL
LIN {X 0,Y 119.967,Z 600.286,A -85,B 0,C 180,E1 -34357.696,E2 -34357.696} C_VEL
LIN {X 0,Y 113.558,Z 593.239,A -85,B 0,C 180,E1 -34364.511,E2 -34364.511} C_VEL
LIN {X 0,Y 111.352,Z 590.349,A -85,B 0,C 180,E1 -34366.847,E2 -34366.847} C_VEL
LIN {X 0,Y 106.816,Z 584.655,A -85,B 0,C 180,E1 -34370.366,E2 -34370.366} C_VEL
LIN {X 0,Y 102.792,Z 578.456,A -85,B 0,C 180,E1 -34374.038,E2 -34374.038} C_VEL
LIN {X 0,Y 101.506,Z 574.718,A -85,B 0,C 180,E1 -34376.575,E2 -34376.575} C_VEL
LIN {X 0,Y 100.669,Z 565.551,A -85,B 0,C 180,E1 -34382.991,E2 -34382.991} C_VEL
LIN {X 0,Y 100.333,Z 556.823,A -85,B 0,C 180,E1 -34388.026,E2 -34388.026} C_VEL
LIN {X 0,Y 100.061,Z 547.178,A -85,B 0,C 180,E1 -34392.636,E2 -34392.636} C_VEL
LIN {X 0,Y 100.064,Z 535.382,A -85,B 0,C 180,E1 -34397.307,E2 -34397.307} C_VEL
LIN {X 0,Y 100.454,Z 522.715,A -85,B 0,C 180,E1 -34401.4,E2 -34401.4} C_VEL
LIN {X 0,Y 101.094,Z 508.92,A -85,B 0,C 180,E1 -34404.96,E2 -34404.96} C_VEL
LIN {X 0,Y 101.865,Z 494.012,A -85,B 0,C 180,E1 -34407.932,E2 -34407.932} C_VEL
LIN {X 0,Y 101.648,Z 496.013,A -85,B 0,C 180,E1 -34408.84,E2 -34408.84} C_VEL
LIN {X 0,Y 102.909,Z 496.246,A -85,B 0,C 180,E1 -34410.696,E2 -34410.696} C_VEL
LIN {X 0,Y 103.935,Z 495.296,A -85,B 0,C 180,E1 -34411.486,E2 -34411.486} C_VEL
LIN {X 0,Y 106.621,Z 491.649,A -85,B 0,C 180,E1 -34412.818,E2 -34412.818} C_VEL
LIN {X 0,Y 108.221,Z 488.86,A -85,B 0,C 180,E1 -34413.377,E2 -34413.377} C_VEL
LIN {X 0,Y 110.117,Z 487.788,A -85,B 0,C 180,E1 -34414.923,E2 -34414.923} C_VEL
LIN {X 0,Y 112.381,Z 485.666,A -85,B 0,C 180,E1 -34416.309,E2 -34416.309} C_VEL
LIN {X 0,Y 115.409,Z 481.434,A -85,B 0,C 180,E1 -34417.641,E2 -34417.641} C_VEL
LIN {X 0,Y 118.972,Z 474.386,A -85,B 0,C 180,E1 -34418.722,E2 -34418.722} C_VEL
LIN {X 0,Y 119.338,Z 473.677,A -85,B 0,C 180,E1 -34418.851,E2 -34418.851} C_VEL
LIN {X 0,Y 121.909,Z 471.318,A -85,B 0,C 180,E1 -34420.269,E2 -34420.269} C_VEL
LIN {X 0,Y 124.927,Z 466.985,A -85,B 0,C 180,E1 -34421.61,E2 -34421.61} C_VEL
LIN {X 0,Y 127.713,Z 461.343,A -85,B 0,C 180,E1 -34422.609,E2 -34422.609} C_VEL
LIN {X 0,Y 131.522,Z 450.55,A -85,B 0,C 180,E1 -34423.815,E2 -34423.815} C_VEL
LIN {X 0,Y 132.59,Z 447.559,A -85,B 0,C 180,E1 -34424.16,E2 -34424.16} C_VEL
LIN {X 0,Y 135.795,Z 443.544,A -85,B 0,C 180,E1 -34425.567,E2 -34425.567} C_VEL
LIN {X 0,Y 139.158,Z 437.617,A -85,B 0,C 180,E1 -34426.795,E2 -34426.795} C_VEL
LIN {X 0,Y 140.412,Z 434.813,A -85,B 0,C 180,E1 -34427.184,E2 -34427.184} C_VEL
LIN {X 0,Y 137.966,Z 463.732,A -85,B 0,C 180,E1 -34428.449,E2 -34428.449} C_VEL
LIN {X 0,Y 135.816,Z 477.73,A -85,B 0,C 180,E1 -34429.488,E2 -34429.488} C_VEL
LIN {X 0,Y 132.856,Z 491.341,A -85,B 0,C 180,E1 -34430.988,E2 -34430.988} C_VEL
LIN {X 0,Y 129.13,Z 504.143,A -85,B 0,C 180,E1 -34432.873,E2 -34432.873} C_VEL
LIN {X 0,Y 124.511,Z 516.664,A -85,B 0,C 180,E1 -34435.27,E2 -34435.27} C_VEL
LIN {X 0,Y 119.799,Z 528.042,A -85,B 0,C 180,E1 -34438.241,E2 -34438.241} C_VEL
LIN {X 0,Y 115.92,Z 536.544,A -85,B 0,C 180,E1 -34441.083,E2 -34441.083} C_VEL
LIN {X 0,Y 110.405,Z 547.294,A -85,B 0,C 180,E1 -34445.636,E2 -34445.636} C_VEL
LIN {X 0,Y 105.617,Z 556.168,A -85,B 0,C 180,E1 -34450.625,E2 -34450.625} C_VEL
LIN {X 0,Y 101.752,Z 563.539,A -85,B 0,C 180,E1 -34456.049,E2 -34456.049} C_VEL
LIN {X 0,Y 98.819,Z 569.682,A -85,B 0,C 180,E1 -34461.84,E2 -34461.84} C_VEL
LIN {X 0,Y 96.554,Z 574.806,A -85,B 0,C 180,E1 -34467.911,E2 -34467.911} C_VEL
LIN {X 0,Y 94.744,Z 580.134,A -85,B 0,C 180,E1 -34476.356,E2 -34476.356} C_VEL
LIN {X 0,Y 94.557,Z 583.14,A -85,B 0,C 180,E1 -34482.829,E2 -34482.829} C_VEL
LIN {X 0,Y 95.724,Z 585.913,A -85,B 0,C 180,E1 -34491.45,E2 -34491.45} C_VEL
LIN {X 0,Y 98.78,Z 587.279,A -85,B 0,C 180,E1 -34499.748,E2 -34499.748} C_VEL
LIN {X 0,Y 103.538,Z 587.28,A -85,B 0,C 180,E1 -34507.494,E2 -34507.494} C_VEL
LIN {X 0,Y 109.89,Z 585.905,A -85,B 0,C 180,E1 -34514.506,E2 -34514.506} C_VEL
LIN {X 0,Y 117.612,Z 583.115,A -85,B 0,C 180,E1 -34520.72,E2 -34520.72} C_VEL
LIN {X 0,Y 126.521,Z 578.815,A -85,B 0,C 180,E1 -34526.127,E2 -34526.127} C_VEL
LIN {X 0,Y 133.854,Z 574.492,A -85,B 0,C 180,E1 -34529.688,E2 -34529.688} C_VEL
LIN {X 0,Y 143.431,Z 567.758,A -85,B 0,C 180,E1 -34533.605,E2 -34533.605} C_VEL
LIN {X 0,Y 152.516,Z 560.174,A -85,B 0,C 180,E1 -34536.692,E2 -34536.692} C_VEL
LIN {X 0,Y 161.109,Z 551.778,A -85,B 0,C 180,E1 -34539.167,E2 -34539.167} C_VEL
LIN {X 0,Y 169.957,Z 541.596,A -85,B 0,C 180,E1 -34541.403,E2 -34541.403} C_VEL
LIN {X 0,Y 178.229,Z 530.103,A -85,B 0,C 180,E1 -34543.302,E2 -34543.302} C_VEL
LIN {X 0,Y 184.98,Z 518.83,A -85,B 0,C 180,E1 -34544.717,E2 -34544.717} C_VEL
LIN {X 0,Y 191.318,Z 505.863,A -85,B 0,C 180,E1 -34545.953,E2 -34545.953} C_VEL
LIN {X 0,Y 196.206,Z 493.131,A -85,B 0,C 180,E1 -34546.91,E2 -34546.91} C_VEL
LIN {X 0,Y 200.355,Z 478.81,A -85,B 0,C 180,E1 -34547.7,E2 -34547.7} C_VEL
LIN {X 0,Y 203.164,Z 464.706,A -85,B 0,C 180,E1 -34548.219,E2 -34548.219} C_VEL
LIN {X 0,Y 203.616,Z 461.259,A -85,B 0,C 180,E1 -34548.34,E2 -34548.34} C_VEL
LIN {X 0,Y 201.307,Z 455.361,A -85,B 0,C 180,E1 -34551.496,E2 -34551.496} C_VEL
LIN {X 0,Y 199.107,Z 450.189,A -85,B 0,C 180,E1 -34555.207,E2 -34555.207} C_VEL
LIN {X 0,Y 197.663,Z 446.638,A -85,B 0,C 180,E1 -34558.731,E2 -34558.731} C_VEL
LIN {X 0,Y 196.666,Z 443.159,A -85,B 0,C 180,E1 -34564.333,E2 -34564.333} C_VEL
LIN {X 0,Y 196.598,Z 443.504,A -85,B 0,C 180,E1 -34566.473,E2 -34566.473} C_VEL
LIN {X 0,Y 196.983,Z 446.232,A -85,B 0,C 180,E1 -34570.5,E2 -34570.5} C_VEL
LIN {X 0,Y 197.705,Z 448.681,A -85,B 0,C 180,E1 -34573.184,E2 -34573.184} C_VEL
LIN {X 0,Y 198.915,Z 453.013,A -85,B 0,C 180,E1 -34576.297,E2 -34576.297} C_VEL
LIN {X 0,Y 200.412,Z 458.209,A -85,B 0,C 180,E1 -34579.151,E2 -34579.151} C_VEL
LIN {X 0,Y 202.015,Z 464.167,A -85,B 0,C 180,E1 -34581.683,E2 -34581.683} C_VEL
LIN {X 0,Y 202.933,Z 468.183,A -85,B 0,C 180,E1 -34583.099,E2 -34583.099} C_VEL
LIN {X 0,Y 200.277,Z 482.878,A -85,B 0,C 180,E1 -34583.503,E2 -34583.503} C_VEL
LIN {X 0,Y 196.36,Z 497.009,A -85,B 0,C 180,E1 -34584.053,E2 -34584.053} C_VEL
LIN {X 0,Y 191.833,Z 509.29,A -85,B 0,C 180,E1 -34584.748,E2 -34584.748} C_VEL
LIN {X 0,Y 185.5,Z 522.581,A -85,B 0,C 180,E1 -34585.656,E2 -34585.656} C_VEL
LIN {X 0,Y 178.51,Z 534.533,A -85,B 0,C 180,E1 -34586.803,E2 -34586.803} C_VEL
LIN {X 0,Y 170.928,Z 545.456,A -85,B 0,C 180,E1 -34588.245,E2 -34588.245} C_VEL
LIN {X 0,Y 161.98,Z 556.264,A -85,B 0,C 180,E1 -34590.148,E2 -34590.148} C_VEL
LIN {X 0,Y 153.362,Z 565.214,A -85,B 0,C 180,E1 -34592.347,E2 -34592.347} C_VEL
LIN {X 0,Y 143.67,Z 573.821,A -85,B 0,C 180,E1 -34595.265,E2 -34595.265} C_VEL
LIN {X 0,Y 134.385,Z 580.801,A -85,B 0,C 180,E1 -34598.584,E2 -34598.584} C_VEL
LIN {X 0,Y 124.573,Z 587.12,A -85,B 0,C 180,E1 -34603.046,E2 -34603.046} C_VEL
LIN {X 0,Y 115.717,Z 591.849,A -85,B 0,C 180,E1 -34608.265,E2 -34608.265} C_VEL
LIN {X 0,Y 108.145,Z 595.137,A -85,B 0,C 180,E1 -34614.355,E2 -34614.355} C_VEL
LIN {X 0,Y 102.063,Z 597.102,A -85,B 0,C 180,E1 -34621.3,E2 -34621.3} C_VEL
LIN {X 0,Y 97.618,Z 597.781,A -85,B 0,C 180,E1 -34628.987,E2 -34628.987} C_VEL
LIN {X 0,Y 95.161,Z 597.187,A -85,B 0,C 180,E1 -34637.254,E2 -34637.254} C_VEL
LIN {X 0,Y 94.75,Z 595.3,A -85,B 0,C 180,E1 -34645.771,E2 -34645.771} C_VEL
LIN {X 0,Y 95.362,Z 593.86,A -85,B 0,C 180,E1 -34650.01,E2 -34650.01} C_VEL
LIN {X 0,Y 96.876,Z 591.041,A -85,B 0,C 180,E1 -34656.236,E2 -34656.236} C_VEL
LIN {X 0,Y 100.022,Z 585.879,A -85,B 0,C 180,E1 -34664.198,E2 -34664.198} C_VEL
LIN {X 0,Y 103.075,Z 581.98,A -85,B 0,C 180,E1 -34668.841,E2 -34668.841} C_VEL
LIN {X 0,Y 106.336,Z 590.823,A -85,B 0,C 180,E1 -34677.468,E2 -34677.468} C_VEL
LIN {X 0,Y 112.715,Z 598.429,A -85,B 0,C 180,E1 -34685.486,E2 -34685.486} C_VEL
LIN {X 0,Y 120.61,Z 604.035,A -85,B 0,C 180,E1 -34691.912,E2 -34691.912} C_VEL
LIN {X 0,Y 131.962,Z 609.164,A -85,B 0,C 180,E1 -34698.007,E2 -34698.007} C_VEL
LIN {X 0,Y 140.008,Z 611.597,A -85,B 0,C 180,E1 -34701.18,E2 -34701.18} C_VEL
LIN {X 0,Y 140.739,Z 611.754,A -85,B 0,C 180,E1 -34701.889,E2 -34701.889} C_VEL
LIN {X 0,Y 130.786,Z 608.154,A -85,B 0,C 180,E1 -34705.782,E2 -34705.782} C_VEL
LIN {X 0,Y 121.487,Z 603.388,A -85,B 0,C 180,E1 -34710.654,E2 -34710.654} C_VEL
LIN {X 0,Y 113.7,Z 597.606,A -85,B 0,C 180,E1 -34716.395,E2 -34716.395} C_VEL
LIN {X 0,Y 107.626,Z 590.71,A -85,B 0,C 180,E1 -34722.97,E2 -34722.97} C_VEL
LIN {X 0,Y 103.474,Z 582.566,A -85,B 0,C 180,E1 -34730.257,E2 -34730.257} C_VEL
LIN {X 0,Y 101.506,Z 574.718,A -85,B 0,C 180,E1 -34736.575,E2 -34736.575} C_VEL
LIN {X 0,Y 100.425,Z 570.913,A -85,B 0,C 180,E1 -34739.052,E2 -34739.052} C_VEL
LIN {X 0,Y 98.722,Z 566.692,A -85,B 0,C 180,E1 -34741.242,E2 -34741.242} C_VEL
LIN {X 0,Y 95.074,Z 557.525,A -85,B 0,C 180,E1 -34745.341,E2 -34745.341} C_VEL
LIN {X 0,Y 93.893,Z 551.268,A -85,B 0,C 180,E1 -34748.317,E2 -34748.317} C_VEL
LIN {X 0,Y 93.538,Z 540.729,A -85,B 0,C 180,E1 -34753.183,E2 -34753.183} C_VEL
LIN {X 0,Y 93.633,Z 528.25,A -85,B 0,C 180,E1 -34757.974,E2 -34757.974} C_VEL
LIN {X 0,Y 94.112,Z 513.79,A -85,B 0,C 180,E1 -34762.422,E2 -34762.422} C_VEL
LIN {X 0,Y 94.412,Z 505.91,A -85,B 0,C 180,E1 -34764.373,E2 -34764.373} C_VEL
LIN {X 0,Y 94.084,Z 507.468,A -85,B 0,C 180,E1 -34765.345,E2 -34765.345} C_VEL
LIN {X 0,Y 94.385,Z 508.015,A -85,B 0,C 180,E1 -34766.44,E2 -34766.44} C_VEL
LIN {X 0,Y 95.467,Z 507.486,A -85,B 0,C 180,E1 -34767.824,E2 -34767.824} C_VEL
LIN {X 0,Y 96.797,Z 506.265,A -85,B 0,C 180,E1 -34768.91,E2 -34768.91} C_VEL
LIN {X 0,Y 98.45,Z 504.379,A -85,B 0,C 180,E1 -34769.87,E2 -34769.87} C_VEL
LIN {X 0,Y 100.489,Z 502.732,A -85,B 0,C 180,E1 -34771.518,E2 -34771.518} C_VEL
LIN {X 0,Y 102.348,Z 501.719,A -85,B 0,C 180,E1 -34773.196,E2 -34773.196} C_VEL
LIN {X 0,Y 104.754,Z 499.442,A -85,B 0,C 180,E1 -34774.636,E2 -34774.636} C_VEL
LIN {X 0,Y 109.036,Z 494.163,A -85,B 0,C 180,E1 -34776.457,E2 -34776.457} C_VEL
LIN {X 0,Y 111.295,Z 492.531,A -85,B 0,C 180,E1 -34777.852,E2 -34777.852} C_VEL
LIN {X 0,Y 113.603,Z 490.301,A -85,B 0,C 180,E1 -34778.956,E2 -34778.956} C_VEL
LIN {X 0,Y 116.742,Z 486.328,A -85,B 0,C 180,E1 -34780.165,E2 -34780.165} C_VEL
LIN {X 0,Y 120.176,Z 480.619,A -85,B 0,C 180,E1 -34781.113,E2 -34781.113} C_VEL
LIN {X 0,Y 121.365,Z 478.555,A -85,B 0,C 180,E1 -34781.447,E2 -34781.447} C_VEL
LIN {X 0,Y 125.048,Z 474.644,A -85,B 0,C 180,E1 -34783.053,E2 -34783.053} C_VEL
LIN {X 0,Y 128.759,Z 469.108,A -85,B 0,C 180,E1 -34784.322,E2 -34784.322} C_VEL
LIN {X 0,Y 132.339,Z 461.571,A -85,B 0,C 180,E1 -34785.336,E2 -34785.336} C_VEL
LIN {X 0,Y 133.964,Z 457.255,A -85,B 0,C 180,E1 -34785.774,E2 -34785.774} C_VEL
LIN {X 0,Y 132.452,Z 470.215,A -85,B 0,C 180,E1 -34786.56,E2 -34786.56} C_VEL
LIN {X 0,Y 129.79,Z 484.458,A -85,B 0,C 180,E1 -34787.869,E2 -34787.869} C_VEL
LIN {X 0,Y 125.974,Z 498.853,A -85,B 0,C 180,E1 -34789.722,E2 -34789.722} C_VEL
LIN {X 0,Y 121.675,Z 511.034,A -85,B 0,C 180,E1 -34791.759,E2 -34791.759} C_VEL
LIN {X 0,Y 116.497,Z 523.583,A -85,B 0,C 180,E1 -34794.631,E2 -34794.631} C_VEL
LIN {X 0,Y 111.375,Z 534.863,A -85,B 0,C 180,E1 -34798.207,E2 -34798.207} C_VEL
LIN {X 0,Y 105.794,Z 545.185,A -85,B 0,C 180,E1 -34802.38,E2 -34802.38} C_VEL
LIN {X 0,Y 100.611,Z 554.472,A -85,B 0,C 180,E1 -34807.476,E2 -34807.476} C_VEL
LIN {X 0,Y 96.08,Z 562.224,A -85,B 0,C 180,E1 -34813.035,E2 -34813.035} C_VEL
LIN {X 0,Y 92.664,Z 568.822,A -85,B 0,C 180,E1 -34819.315,E2 -34819.315} C_VEL
LIN {X 0,Y 90.104,Z 573.964,A -85,B 0,C 180,E1 -34825.531,E2 -34825.531} C_VEL
LIN {X 0,Y 88.232,Z 578.375,A -85,B 0,C 180,E1 -34832.264,E2 -34832.264} C_VEL
LIN {X 0,Y 87.437,Z 581.89,A -85,B 0,C 180,E1 -34839.208,E2 -34839.208} C_VEL
LIN {X 0,Y 88.043,Z 585.275,A -85,B 0,C 180,E1 -34848.544,E2 -34848.544} C_VEL
LIN {X 0,Y 90.49,Z 587.251,A -85,B 0,C 180,E1 -34857.661,E2 -34857.661} C_VEL
LIN {X 0,Y 94.976,Z 587.855,A -85,B 0,C 180,E1 -34866.143,E2 -34866.143} C_VEL
LIN {X 0,Y 101.098,Z 587.101,A -85,B 0,C 180,E1 -34873.841,E2 -34873.841} C_VEL
LIN {X 0,Y 108.792,Z 584.949,A -85,B 0,C 180,E1 -34880.573,E2 -34880.573} C_VEL
LIN {X 0,Y 117.74,Z 581.338,A -85,B 0,C 180,E1 -34886.378,E2 -34886.378} C_VEL
LIN {X 0,Y 124.858,Z 577.721,A -85,B 0,C 180,E1 -34890.064,E2 -34890.064} C_VEL
LIN {X 0,Y 132.966,Z 572.874,A -85,B 0,C 180,E1 -34893.559,E2 -34893.559} C_VEL
LIN {X 0,Y 142.106,Z 566.375,A -85,B 0,C 180,E1 -34896.881,E2 -34896.881} C_VEL
LIN {X 0,Y 151.238,Z 558.71,A -85,B 0,C 180,E1 -34899.674,E2 -34899.674} C_VEL
LIN {X 0,Y 160.516,Z 549.537,A -85,B 0,C 180,E1 -34902.071,E2 -34902.071} C_VEL
LIN {X 0,Y 169.309,Z 539.174,A -85,B 0,C 180,E1 -34904.103,E2 -34904.103} C_VEL
LIN {X 0,Y 177.047,Z 528.258,A -85,B 0,C 180,E1 -34905.736,E2 -34905.736} C_VEL
LIN {X 0,Y 184.254,Z 516.012,A -85,B 0,C 180,E1 -34907.113,E2 -34907.113} C_VEL
LIN {X 0,Y 190.468,Z 502.881,A -85,B 0,C 180,E1 -34908.245,E2 -34908.245} C_VEL
LIN {X 0,Y 195.102,Z 490.322,A -85,B 0,C 180,E1 -34909.073,E2 -34909.073} C_VEL
LIN {X 0,Y 198.983,Z 476.066,A -85,B 0,C 180,E1 -34909.774,E2 -34909.774} C_VEL
LIN {X 0,Y 201.008,Z 465.457,A -85,B 0,C 180,E1 -34910.156,E2 -34910.156} C_VEL
LIN {X 0,Y 199.079,Z 459.959,A -85,B 0,C 180,E1 -34913.434,E2 -34913.434} C_VEL
LIN {X 0,Y 197.535,Z 456.158,A -85,B 0,C 180,E1 -34916.57,E2 -34916.57} C_VEL
LIN {X 0,Y 196.643,Z 453.564,A -85,B 0,C 180,E1 -34919.107,E2 -34919.107} C_VEL
LIN {X 0,Y 195.781,Z 450.474,A -85,B 0,C 180,E1 -34924.103,E2 -34924.103} C_VEL
LIN {X 0,Y 195.712,Z 450.63,A -85,B 0,C 180,E1 -34926.422,E2 -34926.422} C_VEL
LIN {X 0,Y 196.045,Z 453.272,A -85,B 0,C 180,E1 -34930.291,E2 -34930.291} C_VEL
LIN {X 0,Y 196.603,Z 455.428,A -85,B 0,C 180,E1 -34932.604,E2 -34932.604} C_VEL
LIN {X 0,Y 197.645,Z 459.622,A -85,B 0,C 180,E1 -34935.612,E2 -34935.612} C_VEL
LIN {X 0,Y 198.928,Z 464.603,A -85,B 0,C 180,E1 -34938.371,E2 -34938.371} C_VEL
LIN {X 0,Y 200.279,Z 470.924,A -85,B 0,C 180,E1 -34941.007,E2 -34941.007} C_VEL
LIN {X 0,Y 200.376,Z 471.498,A -85,B 0,C 180,E1 -34941.221,E2 -34941.221} C_VEL
LIN {X 0,Y 197.467,Z 485.592,A -85,B 0,C 180,E1 -34941.654,E2 -34941.654} C_VEL
LIN {X 0,Y 193.074,Z 499.931,A -85,B 0,C 180,E1 -34942.224,E2 -34942.224} C_VEL
LIN {X 0,Y 188.172,Z 512.122,A -85,B 0,C 180,E1 -34942.901,E2 -34942.901} C_VEL
LIN {X 0,Y 181.75,Z 524.729,A -85,B 0,C 180,E1 -34943.767,E2 -34943.767} C_VEL
LIN {X 0,Y 174.644,Z 536.223,A -85,B 0,C 180,E1 -34944.864,E2 -34944.864} C_VEL
LIN {X 0,Y 166.161,Z 547.758,A -85,B 0,C 180,E1 -34946.406,E2 -34946.406} C_VEL
LIN {X 0,Y 157.045,Z 558.117,A -85,B 0,C 180,E1 -34948.266,E2 -34948.266} C_VEL
LIN {X 0,Y 148.239,Z 566.69,A -85,B 0,C 180,E1 -34950.435,E2 -34950.435} C_VEL
LIN {X 0,Y 138.285,Z 574.949,A -85,B 0,C 180,E1 -34953.319,E2 -34953.319} C_VEL
LIN {X 0,Y 128.476,Z 581.794,A -85,B 0,C 180,E1 -34956.748,E2 -34956.748} C_VEL
LIN {X 0,Y 119.827,Z 586.978,A -85,B 0,C 180,E1 -34960.557,E2 -34960.557} C_VEL
LIN {X 0,Y 110.515,Z 591.612,A -85,B 0,C 180,E1 -34965.812,E2 -34965.812} C_VEL
LIN {X 0,Y 102.421,Z 594.831,A -85,B 0,C 180,E1 -34972.025,E2 -34972.025} C_VEL
LIN {X 0,Y 95.864,Z 596.733,A -85,B 0,C 180,E1 -34979.251,E2 -34979.251} C_VEL
LIN {X 0,Y 90.879,Z 597.344,A -85,B 0,C 180,E1 -34987.652,E2 -34987.652} C_VEL
LIN {X 0,Y 88.23,Z 596.692,A -85,B 0,C 180,E1 -34996.233,E2 -34996.233} C_VEL
LIN {X 0,Y 87.648,Z 594.74,A -85,B 0,C 180,E1 -35005.428,E2 -35005.428} C_VEL
LIN {X 0,Y 89.26,Z 591.436,A -85,B 0,C 180,E1 -35014.512,E2 -35014.512} C_VEL
LIN {X 0,Y 91.213,Z 587.976,A -85,B 0,C 180,E1 -35021.079,E2 -35021.079} C_VEL
LIN {X 0,Y 95.642,Z 581.903,A -85,B 0,C 180,E1 -35029.253,E2 -35029.253} C_VEL
LIN {X 0,Y 97.462,Z 580.071,A -85,B 0,C 180,E1 -35031.346,E2 -35031.346} C_VEL
LIN {X 0,Y 100.639,Z 587.908,A -85,B 0,C 180,E1 -35039.167,E2 -35039.167} C_VEL
LIN {X 0,Y 106.269,Z 594.841,A -85,B 0,C 180,E1 -35046.396,E2 -35046.396} C_VEL
LIN {X 0,Y 113.596,Z 600.575,A -85,B 0,C 180,E1 -35052.719,E2 -35052.719} C_VEL
LIN {X 0,Y 122.534,Z 605.36,A -85,B 0,C 180,E1 -35058.009,E2 -35058.009} C_VEL
LIN {X 0,Y 128.969,Z 607.945,A -85,B 0,C 180,E1 -35060.915,E2 -35060.915} C_VEL
LIN {X 0,Y 130.067,Z 608.31,A -85,B 0,C 180,E1 -35061.889,E2 -35061.889} C_VEL
LIN {X 0,Y 120.136,Z 603.667,A -85,B 0,C 180,E1 -35066.366,E2 -35066.366} C_VEL
LIN {X 0,Y 110.718,Z 597.408,A -85,B 0,C 180,E1 -35072.354,E2 -35072.354} C_VEL
LIN {X 0,Y 102.76,Z 589.245,A -85,B 0,C 180,E1 -35080.073,E2 -35080.073} C_VEL
LIN {X 0,Y 97.599,Z 579.794,A -85,B 0,C 180,E1 -35088.617,E2 -35088.617} C_VEL
LIN {X 0,Y 95.274,Z 570.613,A -85,B 0,C 180,E1 -35096.091,E2 -35096.091} C_VEL
LIN {X 0,Y 94.49,Z 562.092,A -85,B 0,C 180,E1 -35102.124,E2 -35102.124} C_VEL
LIN {X 0,Y 94.083,Z 554.885,A -85,B 0,C 180,E1 -35106.412,E2 -35106.412} C_VEL
LIN {X 0,Y 93.893,Z 551.268,A -85,B 0,C 180,E1 -35108.317,E2 -35108.317} C_VEL
LIN {X 0,Y 93.182,Z 546.562,A -85,B 0,C 180,E1 -35110.411,E2 -35110.411} C_VEL
LIN {X 0,Y 91.666,Z 541.53,A -85,B 0,C 180,E1 -35112.157,E2 -35112.157} C_VEL
LIN {X 0,Y 88.167,Z 531.096,A -85,B 0,C 180,E1 -35115.232,E2 -35115.232} C_VEL
LIN {X 0,Y 87.191,Z 525.733,A -85,B 0,C 180,E1 -35116.878,E2 -35116.878} C_VEL
LIN {X 0,Y 87.119,Z 523.933,A -85,B 0,C 180,E1 -35117.471,E2 -35117.471} C_VEL
LIN {X 0,Y 87.328,Z 515.79,A -85,B 0,C 180,E1 -35120.16,E2 -35120.16} C_VEL
LIN {X 0,Y 86.864,Z 517.241,A -85,B 0,C 180,E1 -35121.276,E2 -35121.276} C_VEL
LIN {X 0,Y 87.639,Z 517.404,A -85,B 0,C 180,E1 -35123.554,E2 -35123.554} C_VEL
LIN {X 0,Y 91.386,Z 514.267,A -85,B 0,C 180,E1 -35127.379,E2 -35127.379} C_VEL
LIN {X 0,Y 92.926,Z 513.634,A -85,B 0,C 180,E1 -35129.337,E2 -35129.337} C_VEL
LIN {X 0,Y 96.12,Z 511.239,A -85,B 0,C 180,E1 -35131.892,E2 -35131.892} C_VEL
LIN {X 0,Y 97.508,Z 509.829,A -85,B 0,C 180,E1 -35132.599,E2 -35132.599} C_VEL
LIN {X 0,Y 103.018,Z 506.138,A -85,B 0,C 180,E1 -35136.508,E2 -35136.508} C_VEL
LIN {X 0,Y 107.059,Z 502.166,A -85,B 0,C 180,E1 -35138.255,E2 -35138.255} C_VEL
LIN {X 0,Y 108.766,Z 500.059,A -85,B 0,C 180,E1 -35138.808,E2 -35138.808} C_VEL
LIN {X 0,Y 112.723,Z 496.937,A -85,B 0,C 180,E1 -35140.727,E2 -35140.727} C_VEL
LIN {X 0,Y 116.575,Z 493.019,A -85,B 0,C 180,E1 -35142.196,E2 -35142.196} C_VEL
LIN {X 0,Y 120.917,Z 487.222,A -85,B 0,C 180,E1 -35143.381,E2 -35143.381} C_VEL
LIN {X 0,Y 123.696,Z 482.946,A -85,B 0,C 180,E1 -35144.019,E2 -35144.019} C_VEL
LIN {X 0,Y 125.614,Z 481.05,A -85,B 0,C 180,E1 -35144.763,E2 -35144.763} C_VEL
LIN {X 0,Y 125.683,Z 482.868,A -85,B 0,C 180,E1 -35145.209,E2 -35145.209} C_VEL
LIN {X 0,Y 121.922,Z 497.106,A -85,B 0,C 180,E1 -35146.972,E2 -35146.972} C_VEL
LIN {X 0,Y 117.445,Z 509.715,A -85,B 0,C 180,E1 -35148.991,E2 -35148.991} C_VEL
LIN {X 0,Y 111.968,Z 522.585,A -85,B 0,C 180,E1 -35151.837,E2 -35151.837} C_VEL
LIN {X 0,Y 106.485,Z 534.113,A -85,B 0,C 180,E1 -35155.424,E2 -35155.424} C_VEL
LIN {X 0,Y 100.547,Z 544.635,A -85,B 0,C 180,E1 -35159.654,E2 -35159.654} C_VEL
LIN {X 0,Y 94.956,Z 554.1,A -85,B 0,C 180,E1 -35164.892,E2 -35164.892} C_VEL
LIN {X 0,Y 90.009,Z 561.972,A -85,B 0,C 180,E1 -35170.676,E2 -35170.676} C_VEL
LIN {X 0,Y 86.026,Z 569.037,A -85,B 0,C 180,E1 -35177.705,E2 -35177.705} C_VEL
LIN {X 0,Y 82.975,Z 574.748,A -85,B 0,C 180,E1 -35185.146,E2 -35185.146} C_VEL
LIN {X 0,Y 80.662,Z 580.348,A -85,B 0,C 180,E1 -35194.969,E2 -35194.969} C_VEL
LIN {X 0,Y 80.531,Z 584.362,A -85,B 0,C 180,E1 -35205.113,E2 -35205.113} C_VEL
LIN {X 0,Y 82.356,Z 586.953,A -85,B 0,C 180,E1 -35215.153,E2 -35215.153} C_VEL
LIN {X 0,Y 86.41,Z 588.166,A -85,B 0,C 180,E1 -35224.557,E2 -35224.557} C_VEL
LIN {X 0,Y 92.353,Z 588.02,A -85,B 0,C 180,E1 -35233.032,E2 -35233.032} C_VEL
LIN {X 0,Y 99.967,Z 586.497,A -85,B 0,C 180,E1 -35240.404,E2 -35240.404} C_VEL
LIN {X 0,Y 108.936,Z 583.551,A -85,B 0,C 180,E1 -35246.69,E2 -35246.69} C_VEL
LIN {X 0,Y 118.995,Z 579.085,A -85,B 0,C 180,E1 -35251.981,E2 -35251.981} C_VEL
LIN {X 0,Y 127.089,Z 574.594,A -85,B 0,C 180,E1 -35255.4,E2 -35255.4} C_VEL
LIN {X 0,Y 137.773,Z 567.519,A -85,B 0,C 180,E1 -35259.153,E2 -35259.153} C_VEL
LIN {X 0,Y 147.355,Z 559.888,A -85,B 0,C 180,E1 -35261.908,E2 -35261.908} C_VEL
LIN {X 0,Y 155.928,Z 551.857,A -85,B 0,C 180,E1 -35264.013,E2 -35264.013} C_VEL
LIN {X 0,Y 164.312,Z 542.638,A -85,B 0,C 180,E1 -35265.857,E2 -35265.857} C_VEL
LIN {X 0,Y 173.002,Z 531.221,A -85,B 0,C 180,E1 -35267.595,E2 -35267.595} C_VEL
LIN {X 0,Y 179.906,Z 520.316,A -85,B 0,C 180,E1 -35268.849,E2 -35268.849} C_VEL
LIN {X 0,Y 186.684,Z 507.155,A -85,B 0,C 180,E1 -35269.997,E2 -35269.997} C_VEL
LIN {X 0,Y 191.904,Z 494.231,A -85,B 0,C 180,E1 -35270.889,E2 -35270.889} C_VEL
LIN {X 0,Y 196.298,Z 479.749,A -85,B 0,C 180,E1 -35271.619,E2 -35271.619} C_VEL
LIN {X 0,Y 198.488,Z 469.822,A -85,B 0,C 180,E1 -35271.989,E2 -35271.989} C_VEL
LIN {X 0,Y 197.189,Z 465.491,A -85,B 0,C 180,E1 -35274.905,E2 -35274.905} C_VEL
LIN {X 0,Y 196.337,Z 462.973,A -85,B 0,C 180,E1 -35277.03,E2 -35277.03} C_VEL
LIN {X 0,Y 195.55,Z 460.381,A -85,B 0,C 180,E1 -35279.692,E2 -35279.692} C_VEL
LIN {X 0,Y 194.886,Z 457.674,A -85,B 0,C 180,E1 -35284.122,E2 -35284.122} C_VEL
LIN {X 0,Y 194.823,Z 457.817,A -85,B 0,C 180,E1 -35286.451,E2 -35286.451} C_VEL
LIN {X 0,Y 195.107,Z 460.345,A -85,B 0,C 180,E1 -35290.08,E2 -35290.08} C_VEL
LIN {X 0,Y 195.547,Z 462.331,A -85,B 0,C 180,E1 -35292.148,E2 -35292.148} C_VEL
LIN {X 0,Y 196.326,Z 466.208,A -85,B 0,C 180,E1 -35294.925,E2 -35294.925} C_VEL
LIN {X 0,Y 197.28,Z 470.989,A -85,B 0,C 180,E1 -35297.563,E2 -35297.563} C_VEL
LIN {X 0,Y 197.923,Z 475.058,A -85,B 0,C 180,E1 -35299.358,E2 -35299.358} C_VEL
LIN {X 0,Y 194.496,Z 489.453,A -85,B 0,C 180,E1 -35299.78,E2 -35299.78} C_VEL
LIN {X 0,Y 189.965,Z 502.927,A -85,B 0,C 180,E1 -35300.349,E2 -35300.349} C_VEL
LIN {X 0,Y 183.901,Z 516.524,A -85,B 0,C 180,E1 -35301.085,E2 -35301.085} C_VEL
LIN {X 0,Y 177.383,Z 528.205,A -85,B 0,C 180,E1 -35301.898,E2 -35301.898} C_VEL
LIN {X 0,Y 169.432,Z 540.085,A -85,B 0,C 180,E1 -35303.115,E2 -35303.115} C_VEL
LIN {X 0,Y 161.572,Z 549.953,A -85,B 0,C 180,E1 -35304.458,E2 -35304.458} C_VEL
LIN {X 0,Y 152.277,Z 559.823,A -85,B 0,C 180,E1 -35306.255,E2 -35306.255} C_VEL
LIN {X 0,Y 141.818,Z 569.276,A -85,B 0,C 180,E1 -35308.772,E2 -35308.772} C_VEL
LIN {X 0,Y 131.649,Z 576.96,A -85,B 0,C 180,E1 -35311.664,E2 -35311.664} C_VEL
LIN {X 0,Y 121.778,Z 583.244,A -85,B 0,C 180,E1 -35315.112,E2 -35315.112} C_VEL
LIN {X 0,Y 112.78,Z 588.076,A -85,B 0,C 180,E1 -35319.088,E2 -35319.088} C_VEL
LIN {X 0,Y 105.521,Z 591.372,A -85,B 0,C 180,E1 -35323.113,E2 -35323.113} C_VEL
LIN {X 0,Y 96.889,Z 594.526,A -85,B 0,C 180,E1 -35329.424,E2 -35329.424} C_VEL
LIN {X 0,Y 89.819,Z 596.365,A -85,B 0,C 180,E1 -35336.928,E2 -35336.928} C_VEL
LIN {X 0,Y 84.047,Z 596.903,A -85,B 0,C 180,E1 -35346.454,E2 -35346.454} C_VEL
LIN {X 0,Y 81.322,Z 596.196,A -85,B 0,C 180,E1 -35355.038,E2 -35355.038} C_VEL
LIN {X 0,Y 80.553,Z 594.181,A -85,B 0,C 180,E1 -35365.024,E2 -35365.024} C_VEL
LIN {X 0,Y 81.162,Z 592.678,A -85,B 0,C 180,E1 -35370.012,E2 -35370.012} C_VEL
LIN {X 0,Y 82.856,Z 589.759,A -85,B 0,C 180,E1 -35377.297,E2 -35377.297} C_VEL
LIN {X 0,Y 86.407,Z 584.421,A -85,B 0,C 180,E1 -35386.494,E2 -35386.494} C_VEL
LIN {X 0,Y 90.69,Z 579.388,A -85,B 0,C 180,E1 -35392.728,E2 -35392.728} C_VEL
LIN {X 0,Y 92.107,Z 578.019,A -85,B 0,C 180,E1 -35394.138,E2 -35394.138} C_VEL
LIN {X 0,Y 96.452,Z 586.753,A -85,B 0,C 180,E1 -35403.013,E2 -35403.013} C_VEL
LIN {X 0,Y 102.853,Z 593.7,A -85,B 0,C 180,E1 -35410.325,E2 -35410.325} C_VEL
LIN {X 0,Y 110.98,Z 599.524,A -85,B 0,C 180,E1 -35416.548,E2 -35416.548} C_VEL
LIN {X 0,Y 119.163,Z 603.772,A -85,B 0,C 180,E1 -35420.962,E2 -35420.962} C_VEL
LIN {X 0,Y 119.72,Z 603.996,A -85,B 0,C 180,E1 -35421.922,E2 -35421.922} C_VEL
LIN {X 0,Y 109.809,Z 598.193,A -85,B 0,C 180,E1 -35427.167,E2 -35427.167} C_VEL
LIN {X 0,Y 101.635,Z 591.467,A -85,B 0,C 180,E1 -35433.384,E2 -35433.384} C_VEL
LIN {X 0,Y 94.624,Z 582.564,A -85,B 0,C 180,E1 -35441.663,E2 -35441.663} C_VEL
LIN {X 0,Y 90.662,Z 573.179,A -85,B 0,C 180,E1 -35449.989,E2 -35449.989} C_VEL
LIN {X 0,Y 88.827,Z 563.344,A -85,B 0,C 180,E1 -35457.74,E2 -35457.74} C_VEL
LIN {X 0,Y 88.118,Z 554.798,A -85,B 0,C 180,E1 -35463.418,E2 -35463.418} C_VEL
LIN {X 0,Y 87.515,Z 545.16,A -85,B 0,C 180,E1 -35468.631,E2 -35468.631} C_VEL
LIN {X 0,Y 87.062,Z 531.639,A -85,B 0,C 180,E1 -35474.619,E2 -35474.619} C_VEL
LIN {X 0,Y 87.119,Z 523.933,A -85,B 0,C 180,E1 -35477.471,E2 -35477.471} C_VEL
LIN {X 0,Y 87.065,Z 522.082,A -85,B 0,C 180,E1 -35478.568,E2 -35478.568} C_VEL
LIN {X 0,Y 86.948,Z 520.571,A -85,B 0,C 180,E1 -35480.918,E2 -35480.918} C_VEL
LIN {X 0,Y 87.044,Z 520.127,A -85,B 0,C 180,E1 -35483.556,E2 -35483.556} C_VEL
LIN {X 0,Y 88.311,Z 520.21,A -85,B 0,C 180,E1 -35488.323,E2 -35488.323} C_VEL
LIN {X 0,Y 90.115,Z 519.577,A -85,B 0,C 180,E1 -35490.841,E2 -35490.841} C_VEL
LIN {X 0,Y 91.682,Z 518.759,A -85,B 0,C 180,E1 -35492.33,E2 -35492.33} C_VEL
LIN {X 0,Y 95.196,Z 516.36,A -85,B 0,C 180,E1 -35494.767,E2 -35494.767} C_VEL
LIN {X 0,Y 96.615,Z 515.103,A -85,B 0,C 180,E1 -35495.449,E2 -35495.449} C_VEL
LIN {X 0,Y 101.302,Z 512.282,A -85,B 0,C 180,E1 -35498.484,E2 -35498.484} C_VEL
LIN {X 0,Y 105.629,Z 508.827,A -85,B 0,C 180,E1 -35500.379,E2 -35500.379} C_VEL
LIN {X 0,Y 110.163,Z 504.345,A -85,B 0,C 180,E1 -35501.883,E2 -35501.883} C_VEL
LIN {X 0,Y 114.324,Z 501.148,A -85,B 0,C 180,E1 -35503.573,E2 -35503.573} C_VEL
LIN {X 0,Y 115.803,Z 499.78,A -85,B 0,C 180,E1 -35504.077,E2 -35504.077} C_VEL
LIN {X 0,Y 116.121,Z 501.578,A -85,B 0,C 180,E1 -35504.947,E2 -35504.947} C_VEL
LIN {X 0,Y 110.897,Z 514.651,A -85,B 0,C 180,E1 -35507.224,E2 -35507.224} C_VEL
LIN {X 0,Y 105.297,Z 526.616,A -85,B 0,C 180,E1 -35510.177,E2 -35510.177} C_VEL
LIN {X 0,Y 100.108,Z 536.532,A -85,B 0,C 180,E1 -35513.495,E2 -35513.495} C_VEL
LIN {X 0,Y 93.476,Z 547.489,A -85,B 0,C 180,E1 -35518.352,E2 -35518.352} C_VEL
LIN {X 0,Y 87.577,Z 556.539,A -85,B 0,C 180,E1 -35523.891,E2 -35523.891} C_VEL
LIN {X 0,Y 82.65,Z 564.063,A -85,B 0,C 180,E1 -35530.172,E2 -35530.172} C_VEL
LIN {X 0,Y 78.825,Z 570.337,A -85,B 0,C 180,E1 -35537.149,E2 -35537.149} C_VEL
LIN {X 0,Y 75.838,Z 575.534,A -85,B 0,C 180,E1 -35544.688,E2 -35544.688} C_VEL
LIN {X 0,Y 73.866,Z 579.782,A -85,B 0,C 180,E1 -35552.704,E2 -35552.704} C_VEL
LIN {X 0,Y 73.234,Z 583.174,A -85,B 0,C 180,E1 -35561.014,E2 -35561.014} C_VEL
LIN {X 0,Y 73.803,Z 585.438,A -85,B 0,C 180,E1 -35568.365,E2 -35568.365} C_VEL
LIN {X 0,Y 75.822,Z 587.471,A -85,B 0,C 180,E1 -35577.495,E2 -35577.495} C_VEL
LIN {X 0,Y 80.514,Z 588.61,A -85,B 0,C 180,E1 -35587.5,E2 -35587.5} C_VEL
LIN {X 0,Y 87.133,Z 588.392,A -85,B 0,C 180,E1 -35596.326,E2 -35596.326} C_VEL
LIN {X 0,Y 96.313,Z 586.592,A -85,B 0,C 180,E1 -35604.422,E2 -35604.422} C_VEL
LIN {X 0,Y 105.094,Z 583.774,A -85,B 0,C 180,E1 -35610.028,E2 -35610.028} C_VEL
LIN {X 0,Y 115.74,Z 579.205,A -85,B 0,C 180,E1 -35615.178,E2 -35615.178} C_VEL
LIN {X 0,Y 124.22,Z 574.66,A -85,B 0,C 180,E1 -35618.472,E2 -35618.472} C_VEL
LIN {X 0,Y 134.47,Z 568.087,A -85,B 0,C 180,E1 -35621.788,E2 -35621.788} C_VEL
LIN {X 0,Y 145.246,Z 559.716,A -85,B 0,C 180,E1 -35624.657,E2 -35624.657} C_VEL
LIN {X 0,Y 154.878,Z 550.767,A -85,B 0,C 180,E1 -35626.786,E2 -35626.786} C_VEL
LIN {X 0,Y 164.295,Z 540.266,A -85,B 0,C 180,E1 -35628.65,E2 -35628.65} C_VEL
LIN {X 0,Y 173.04,Z 528.454,A -85,B 0,C 180,E1 -35630.233,E2 -35630.233} C_VEL
LIN {X 0,Y 180.605,Z 516.015,A -85,B 0,C 180,E1 -35631.441,E2 -35631.441} C_VEL
LIN {X 0,Y 186.379,Z 504.191,A -85,B 0,C 180,E1 -35632.354,E2 -35632.354} C_VEL
LIN {X 0,Y 191.249,Z 491.628,A -85,B 0,C 180,E1 -35633.104,E2 -35633.104} C_VEL
LIN {X 0,Y 195.369,Z 477.286,A -85,B 0,C 180,E1 -35633.747,E2 -35633.747} C_VEL
LIN {X 0,Y 196.014,Z 474.228,A -85,B 0,C 180,E1 -35633.9,E2 -35633.9} C_VEL
LIN {X 0,Y 194.927,Z 469.851,A -85,B 0,C 180,E1 -35637.392,E2 -35637.392} C_VEL
LIN {X 0,Y 194.302,Z 467.184,A -85,B 0,C 180,E1 -35640.258,E2 -35640.258} C_VEL
LIN {X 0,Y 193.897,Z 464.817,A -85,B 0,C 180,E1 -35644.143,E2 -35644.143} C_VEL
LIN {X 0,Y 193.842,Z 464.991,A -85,B 0,C 180,E1 -35646.484,E2 -35646.484} C_VEL
LIN {X 0,Y 194.042,Z 467.386,A -85,B 0,C 180,E1 -35649.873,E2 -35649.873} C_VEL
LIN {X 0,Y 194.298,Z 469.059,A -85,B 0,C 180,E1 -35651.568,E2 -35651.568} C_VEL
LIN {X 0,Y 194.751,Z 472.38,A -85,B 0,C 180,E1 -35654.02,E2 -35654.02} C_VEL
LIN {X 0,Y 195.403,Z 477.386,A -85,B 0,C 180,E1 -35656.799,E2 -35656.799} C_VEL
LIN {X 0,Y 195.52,Z 478.657,A -85,B 0,C 180,E1 -35657.392,E2 -35657.392} C_VEL
LIN {X 0,Y 192.554,Z 490.24,A -85,B 0,C 180,E1 -35657.775,E2 -35657.775} C_VEL
LIN {X 0,Y 188.408,Z 502.252,A -85,B 0,C 180,E1 -35658.231,E2 -35658.231} C_VEL
LIN {X 0,Y 182.305,Z 515.844,A -85,B 0,C 180,E1 -35658.911,E2 -35658.911} C_VEL
LIN {X 0,Y 174.872,Z 528.859,A -85,B 0,C 180,E1 -35659.751,E2 -35659.751} C_VEL
LIN {X 0,Y 166.785,Z 540.555,A -85,B 0,C 180,E1 -35660.883,E2 -35660.883} C_VEL
LIN {X 0,Y 157.181,Z 552.054,A -85,B 0,C 180,E1 -35662.398,E2 -35662.398} C_VEL
LIN {X 0,Y 147.729,Z 561.507,A -85,B 0,C 180,E1 -35664.134,E2 -35664.134} C_VEL
LIN {X 0,Y 137.024,Z 570.57,A -85,B 0,C 180,E1 -35666.565,E2 -35666.565} C_VEL
LIN {X 0,Y 128.059,Z 576.963,A -85,B 0,C 180,E1 -35668.955,E2 -35668.955} C_VEL
LIN {X 0,Y 119.392,Z 582.265,A -85,B 0,C 180,E1 -35671.731,E2 -35671.731} C_VEL
LIN {X 0,Y 108.443,Z 587.913,A -85,B 0,C 180,E1 -35676.175,E2 -35676.175} C_VEL
LIN {X 0,Y 100.775,Z 591.134,A -85,B 0,C 180,E1 -35680.148,E2 -35680.148} C_VEL
LIN {X 0,Y 91.584,Z 594.221,A -85,B 0,C 180,E1 -35686.518,E2 -35686.518} C_VEL
LIN {X 0,Y 83.925,Z 595.996,A -85,B 0,C 180,E1 -35694.267,E2 -35694.267} C_VEL
LIN {X 0,Y 78.068,Z 596.488,A -85,B 0,C 180,E1 -35703.36,E2 -35703.36} C_VEL
LIN {X 0,Y 74.458,Z 595.701,A -85,B 0,C 180,E1 -35713.621,E2 -35713.621} C_VEL
LIN {X 0,Y 73.465,Z 593.622,A -85,B 0,C 180,E1 -35724.542,E2 -35724.542} C_VEL
LIN {X 0,Y 75.13,Z 590.189,A -85,B 0,C 180,E1 -35735.362,E2 -35735.362} C_VEL
LIN {X 0,Y 77.442,Z 586.595,A -85,B 0,C 180,E1 -35743.081,E2 -35743.081} C_VEL
LIN {X 0,Y 82.47,Z 580.371,A -85,B 0,C 180,E1 -35752.482,E2 -35752.482} C_VEL
LIN {X 0,Y 86.998,Z 575.894,A -85,B 0,C 180,E1 -35757.264,E2 -35757.264} C_VEL
LIN {X 0,Y 92.708,Z 585.476,A -85,B 0,C 180,E1 -35767.2,E2 -35767.2} C_VEL
LIN {X 0,Y 101.438,Z 593.59,A -85,B 0,C 180,E1 -35775.661,E2 -35775.661} C_VEL
LIN {X 0,Y 108.918,Z 598.409,A -85,B 0,C 180,E1 -35780.521,E2 -35780.521} C_VEL
LIN {X 0,Y 109.85,Z 598.864,A -85,B 0,C 180,E1 -35781.955,E2 -35781.955} C_VEL
LIN {X 0,Y 99.372,Z 591.334,A -85,B 0,C 180,E1 -35788.603,E2 -35788.603} C_VEL
LIN {X 0,Y 90.756,Z 581.845,A -85,B 0,C 180,E1 -35797.3,E2 -35797.3} C_VEL
LIN {X 0,Y 85.454,Z 571.232,A -85,B 0,C 180,E1 -35806.973,E2 -35806.973} C_VEL
LIN {X 0,Y 83.139,Z 561.276,A -85,B 0,C 180,E1 -35815.167,E2 -35815.167} C_VEL
LIN {X 0,Y 82.195,Z 552.599,A -85,B 0,C 180,E1 -35821.221,E2 -35821.221} C_VEL
LIN {X 0,Y 81.345,Z 542.825,A -85,B 0,C 180,E1 -35826.8,E2 -35826.8} C_VEL
LIN {X 0,Y 80.748,Z 529.823,A -85,B 0,C 180,E1 -35832.801,E2 -35832.801} C_VEL
LIN {X 0,Y 80.69,Z 524.43,A -85,B 0,C 180,E1 -35834.983,E2 -35834.983} C_VEL
LIN {X 0,Y 80.137,Z 525.475,A -85,B 0,C 180,E1 -35835.917,E2 -35835.917} C_VEL
LIN {X 0,Y 81.332,Z 525.205,A -85,B 0,C 180,E1 -35840.15,E2 -35840.15} C_VEL
LIN {X 0,Y 83.126,Z 523.489,A -85,B 0,C 180,E1 -35842.015,E2 -35842.015} C_VEL
LIN {X 0,Y 84.189,Z 523.392,A -85,B 0,C 180,E1 -35844.582,E2 -35844.582} C_VEL
LIN {X 0,Y 85.83,Z 522.427,A -85,B 0,C 180,E1 -35846.672,E2 -35846.672} C_VEL
LIN {X 0,Y 87.861,Z 520.893,A -85,B 0,C 180,E1 -35848.576,E2 -35848.576} C_VEL
LIN {X 0,Y 90.115,Z 519.577,A -85,B 0,C 180,E1 -35850.841,E2 -35850.841} C_VEL
LIN {X 0,Y 92.731,Z 518.812,A -85,B 0,C 180,E1 -35853.786,E2 -35853.786} C_VEL
LIN {X 0,Y 98.147,Z 518.496,A -85,B 0,C 180,E1 -35859.54,E2 -35859.54} C_VEL
LIN {X 0,Y 101.013,Z 517.244,A -85,B 0,C 180,E1 -35861.326,E2 -35861.326} C_VEL
LIN {X 0,Y 101.469,Z 516.943,A -85,B 0,C 180,E1 -35861.53,E2 -35861.53} C_VEL
LIN {X 0,Y 105.456,Z 514.017,A -85,B 0,C 180,E1 -35863.049,E2 -35863.049} C_VEL
LIN {X 0,Y 107.127,Z 513.406,A -85,B 0,C 180,E1 -35863.997,E2 -35863.997} C_VEL
LIN {X 0,Y 101.234,Z 525.728,A -85,B 0,C 180,E1 -35866.889,E2 -35866.889} C_VEL
LIN {X 0,Y 95.102,Z 536.853,A -85,B 0,C 180,E1 -35870.549,E2 -35870.549} C_VEL
LIN {X 0,Y 88.607,Z 547.015,A -85,B 0,C 180,E1 -35875.019,E2 -35875.019} C_VEL
LIN {X 0,Y 82.262,Z 556.207,A -85,B 0,C 180,E1 -35880.672,E2 -35880.672} C_VEL
LIN {X 0,Y 76.796,Z 563.868,A -85,B 0,C 180,E1 -35887.179,E2 -35887.179} C_VEL
LIN {X 0,Y 71.897,Z 571.163,A -85,B 0,C 180,E1 -35895.887,E2 -35895.887} C_VEL
LIN {X 0,Y 68.705,Z 576.32,A -85,B 0,C 180,E1 -35904.134,E2 -35904.134} C_VEL
LIN {X 0,Y 66.689,Z 580.484,A -85,B 0,C 180,E1 -35912.996,E2 -35912.996} C_VEL
LIN {X 0,Y 66.154,Z 583.799,A -85,B 0,C 180,E1 -35922.21,E2 -35922.21} C_VEL
LIN {X 0,Y 66.814,Z 585.784,A -85,B 0,C 180,E1 -35929.35,E2 -35929.35} C_VEL
LIN {X 0,Y 69.462,Z 587.985,A -85,B 0,C 180,E1 -35940.261,E2 -35940.261} C_VEL
LIN {X 0,Y 74.873,Z 589.051,A -85,B 0,C 180,E1 -35950.891,E2 -35950.891} C_VEL
LIN {X 0,Y 82.26,Z 588.763,A -85,B 0,C 180,E1 -35960.008,E2 -35960.008} C_VEL
LIN {X 0,Y 91.446,Z 587.07,A -85,B 0,C 180,E1 -35967.576,E2 -35967.576} C_VEL
LIN {X 0,Y 101.635,Z 583.996,A -85,B 0,C 180,E1 -35973.604,E2 -35973.604} C_VEL
LIN {X 0,Y 112.862,Z 579.313,A -85,B 0,C 180,E1 -35978.554,E2 -35978.554} C_VEL
LIN {X 0,Y 121.724,Z 574.725,A -85,B 0,C 180,E1 -35981.679,E2 -35981.679} C_VEL
LIN {X 0,Y 131.423,Z 568.679,A -85,B 0,C 180,E1 -35984.545,E2 -35984.545} C_VEL
LIN {X 0,Y 141.893,Z 560.889,A -85,B 0,C 180,E1 -35987.112,E2 -35987.112} C_VEL
LIN {X 0,Y 151.193,Z 552.652,A -85,B 0,C 180,E1 -35989.01,E2 -35989.01} C_VEL
LIN {X 0,Y 159.728,Z 543.708,A -85,B 0,C 180,E1 -35990.593,E2 -35990.593} C_VEL
LIN {X 0,Y 167.976,Z 533.482,A -85,B 0,C 180,E1 -35991.986,E2 -35991.986} C_VEL
LIN {X 0,Y 175.279,Z 522.661,A -85,B 0,C 180,E1 -35993.115,E2 -35993.115} C_VEL
LIN {X 0,Y 182.18,Z 510.228,A -85,B 0,C 180,E1 -35994.117,E2 -35994.117} C_VEL
LIN {X 0,Y 188.076,Z 496.677,A -85,B 0,C 180,E1 -35994.958,E2 -35994.958} C_VEL
LIN {X 0,Y 192.572,Z 483.006,A -85,B 0,C 180,E1 -35995.586,E2 -35995.586} C_VEL
LIN {X 0,Y 193.66,Z 478.939,A -85,B 0,C 180,E1 -35995.766,E2 -35995.766} C_VEL
LIN {X 0,Y 193.022,Z 475.609,A -85,B 0,C 180,E1 -35998.83,E2 -35998.83} C_VEL
LIN {X 0,Y 192.784,Z 473.947,A -85,B 0,C 180,E1 -36000.781,E2 -36000.781} C_VEL
LIN {X 0,Y 192.623,Z 471.888,A -85,B 0,C 180,E1 -36004.171,E2 -36004.171} C_VEL
LIN {X 0,Y 192.576,Z 472.117,A -85,B 0,C 180,E1 -36006.527,E2 -36006.527} C_VEL
LIN {X 0,Y 192.65,Z 474.282,A -85,B 0,C 180,E1 -36009.549,E2 -36009.549} C_VEL
LIN {X 0,Y 192.764,Z 475.82,A -85,B 0,C 180,E1 -36011.067,E2 -36011.067} C_VEL
LIN {X 0,Y 192.985,Z 479.05,A -85,B 0,C 180,E1 -36013.444,E2 -36013.444} C_VEL
LIN {X 0,Y 193.248,Z 482.457,A -85,B 0,C 180,E1 -36015.428,E2 -36015.428} C_VEL
LIN {X 0,Y 189.905,Z 493.848,A -85,B 0,C 180,E1 -36015.801,E2 -36015.801} C_VEL
LIN {X 0,Y 184.88,Z 506.933,A -85,B 0,C 180,E1 -36016.325,E2 -36016.325} C_VEL
LIN {X 0,Y 178.456,Z 519.893,A -85,B 0,C 180,E1 -36016.94,E2 -36016.94} C_VEL
LIN {X 0,Y 170.964,Z 532.05,A -85,B 0,C 180,E1 -36017.741,E2 -36017.741} C_VEL
LIN {X 0,Y 162.767,Z 543.1,A -85,B 0,C 180,E1 -36018.806,E2 -36018.806} C_VEL
LIN {X 0,Y 152.982,Z 554.016,A -85,B 0,C 180,E1 -36020.201,E2 -36020.201} C_VEL
LIN {X 0,Y 143.398,Z 563.055,A -85,B 0,C 180,E1 -36021.884,E2 -36021.884} C_VEL
LIN {X 0,Y 132.45,Z 571.737,A -85,B 0,C 180,E1 -36024.203,E2 -36024.203} C_VEL
LIN {X 0,Y 121.746,Z 578.786,A -85,B 0,C 180,E1 -36026.924,E2 -36026.924} C_VEL
LIN {X 0,Y 111.673,Z 584.319,A -85,B 0,C 180,E1 -36030.118,E2 -36030.118} C_VEL
LIN {X 0,Y 101.647,Z 588.88,A -85,B 0,C 180,E1 -36034.236,E2 -36034.236} C_VEL
LIN {X 0,Y 91.287,Z 592.58,A -85,B 0,C 180,E1 -36039.906,E2 -36039.906} C_VEL
LIN {X 0,Y 82.212,Z 594.936,A -85,B 0,C 180,E1 -36047.048,E2 -36047.048} C_VEL
LIN {X 0,Y 74.724,Z 596,A -85,B 0,C 180,E1 -36055.793,E2 -36055.793} C_VEL
LIN {X 0,Y 69.389,Z 595.792,A -85,B 0,C 180,E1 -36066.201,E2 -36066.201} C_VEL
LIN {X 0,Y 66.678,Z 594.301,A -85,B 0,C 180,E1 -36077.887,E2 -36077.887} C_VEL
LIN {X 0,Y 66.933,Z 591.495,A -85,B 0,C 180,E1 -36090.015,E2 -36090.015} C_VEL
LIN {X 0,Y 68.851,Z 588.445,A -85,B 0,C 180,E1 -36098.792,E2 -36098.792} C_VEL
LIN {X 0,Y 73.001,Z 582.965,A -85,B 0,C 180,E1 -36109.637,E2 -36109.637} C_VEL
LIN {X 0,Y 77.888,Z 577.766,A -85,B 0,C 180,E1 -36116.735,E2 -36116.735} C_VEL
LIN {X 0,Y 82.342,Z 573.717,A -85,B 0,C 180,E1 -36120.898,E2 -36120.898} C_VEL
LIN {X 0,Y 87.775,Z 582.156,A -85,B 0,C 180,E1 -36129.686,E2 -36129.686} C_VEL
LIN {X 0,Y 95.464,Z 589.489,A -85,B 0,C 180,E1 -36137.214,E2 -36137.214} C_VEL
LIN {X 0,Y 99.977,Z 592.747,A -85,B 0,C 180,E1 -36140.428,E2 -36140.428} C_VEL
LIN {X 0,Y 101.318,Z 593.614,A -85,B 0,C 180,E1 -36141.523,E2 -36141.523} C_VEL
LIN {X 0,Y 90.697,Z 584.686,A -85,B 0,C 180,E1 -36149.296,E2 -36149.296} C_VEL
LIN {X 0,Y 83.554,Z 575.41,A -85,B 0,C 180,E1 -36157.837,E2 -36157.837} C_VEL
LIN {X 0,Y 79.078,Z 565.069,A -85,B 0,C 180,E1 -36167.206,E2 -36167.206} C_VEL
LIN {X 0,Y 77.189,Z 555.79,A -85,B 0,C 180,E1 -36174.793,E2 -36174.793} C_VEL
LIN {X 0,Y 76.125,Z 547.256,A -85,B 0,C 180,E1 -36180.659,E2 -36180.659} C_VEL
LIN {X 0,Y 75.035,Z 536.33,A -85,B 0,C 180,E1 -36186.701,E2 -36186.701} C_VEL
LIN {X 0,Y 74.701,Z 532.208,A -85,B 0,C 180,E1 -36188.764,E2 -36188.764} C_VEL
LIN {X 0,Y 74.154,Z 532.955,A -85,B 0,C 180,E1 -36189.515,E2 -36189.515} C_VEL
LIN {X 0,Y 73.777,Z 533.527,A -85,B 0,C 180,E1 -36190.946,E2 -36190.946} C_VEL
LIN {X 0,Y 75.647,Z 531.801,A -85,B 0,C 180,E1 -36196.128,E2 -36196.128} C_VEL
LIN {X 0,Y 77.471,Z 530.974,A -85,B 0,C 180,E1 -36201.202,E2 -36201.202} C_VEL
LIN {X 0,Y 84.089,Z 527.309,A -85,B 0,C 180,E1 -36209.986,E2 -36209.986} C_VEL
LIN {X 0,Y 90.529,Z 523.733,A -85,B 0,C 180,E1 -36215.471,E2 -36215.471} C_VEL
LIN {X 0,Y 94.345,Z 521.356,A -85,B 0,C 180,E1 -36217.771,E2 -36217.771} C_VEL
LIN {X 0,Y 95.821,Z 520.163,A -85,B 0,C 180,E1 -36218.414,E2 -36218.414} C_VEL
LIN {X 0,Y 101.469,Z 516.943,A -85,B 0,C 180,E1 -36221.53,E2 -36221.53} C_VEL
LIN {X 0,Y 100.803,Z 518.121,A -85,B 0,C 180,E1 -36221.701,E2 -36221.701} C_VEL
LIN {X 0,Y 96.274,Z 522.691,A -85,B 0,C 180,E1 -36220.754,E2 -36220.754} C_VEL
LIN {X 0,Y 90.609,Z 527.484,A -85,B 0,C 180,E1 -36218.965,E2 -36218.965} C_VEL
LIN {X 0,Y 87.19,Z 529.686,A -85,B 0,C 180,E1 -36217.216,E2 -36217.216} C_VEL
LIN {X 0,Y 86.56,Z 529.994,A -85,B 0,C 180,E1 -36216.767,E2 -36216.767} C_VEL
LIN {X 0,Y 80.326,Z 533.133,A -85,B 0,C 180,E1 -36211.547,E2 -36211.547} C_VEL
LIN {X 0,Y 73.388,Z 536.543,A -85,B 0,C 180,E1 -36202.443,E2 -36202.443} C_VEL
LIN {X 0,Y 71.318,Z 537.479,A -85,B 0,C 180,E1 -36197.136,E2 -36197.136} C_VEL
LIN {X 0,Y 68.315,Z 540.334,A -85,B 0,C 180,E1 -36185.885,E2 -36185.885} C_VEL
LIN {X 0,Y 68.571,Z 540.346,A -85,B 0,C 180,E1 -36182.927,E2 -36182.927} C_VEL
LIN {X 0,Y 69.697,Z 539.266,A -85,B 0,C 180,E1 -36181.26,E2 -36181.26} C_VEL
LIN {X 0,Y 70.976,Z 547.872,A -85,B 0,C 180,E1 -36175.757,E2 -36175.757} C_VEL
LIN {X 0,Y 72.22,Z 555.161,A -85,B 0,C 180,E1 -36170.228,E2 -36170.228} C_VEL
LIN {X 0,Y 75.392,Z 565.651,A -85,B 0,C 180,E1 -36161.024,E2 -36161.024} C_VEL
LIN {X 0,Y 81.15,Z 575.685,A -85,B 0,C 180,E1 -36151.658,E2 -36151.658} C_VEL
LIN {X 0,Y 90.256,Z 585.382,A -85,B 0,C 180,E1 -36143.026,E2 -36143.026} C_VEL
LIN {X 0,Y 92.347,Z 587.172,A -85,B 0,C 180,E1 -36141.553,E2 -36141.553} C_VEL
LIN {X 0,Y 91.261,Z 586.331,A -85,B 0,C 180,E1 -36140.147,E2 -36140.147} C_VEL
LIN {X 0,Y 83.104,Z 578.657,A -85,B 0,C 180,E1 -36132.414,E2 -36132.414} C_VEL
LIN {X 0,Y 77.886,Z 571.481,A -85,B 0,C 180,E1 -36124.749,E2 -36124.749} C_VEL
LIN {X 0,Y 71.658,Z 576.958,A -85,B 0,C 180,E1 -36119.273,E2 -36119.273} C_VEL
LIN {X 0,Y 66.414,Z 582.239,A -85,B 0,C 180,E1 -36111.678,E2 -36111.678} C_VEL
LIN {X 0,Y 61.88,Z 587.789,A -85,B 0,C 180,E1 -36099.791,E2 -36099.791} C_VEL
LIN {X 0,Y 59.829,Z 590.904,A -85,B 0,C 180,E1 -36090.016,E2 -36090.016} C_VEL
LIN {X 0,Y 59.732,Z 593.773,A -85,B 0,C 180,E1 -36076.453,E2 -36076.453} C_VEL
LIN {X 0,Y 62.938,Z 595.327,A -85,B 0,C 180,E1 -36063.584,E2 -36063.584} C_VEL
LIN {X 0,Y 68.947,Z 595.601,A -85,B 0,C 180,E1 -36052.462,E2 -36052.462} C_VEL
LIN {X 0,Y 77.141,Z 594.602,A -85,B 0,C 180,E1 -36043.434,E2 -36043.434} C_VEL
LIN {X 0,Y 86.889,Z 592.315,A -85,B 0,C 180,E1 -36036.3,E2 -36036.3} C_VEL
LIN {X 0,Y 97.829,Z 588.686,A -85,B 0,C 180,E1 -36030.796,E2 -36030.796} C_VEL
LIN {X 0,Y 109.536,Z 583.605,A -85,B 0,C 180,E1 -36026.481,E2 -36026.481} C_VEL
LIN {X 0,Y 121.823,Z 576.926,A -85,B 0,C 180,E1 -36023.104,E2 -36023.104} C_VEL
LIN {X 0,Y 132.892,Z 569.546,A -85,B 0,C 180,E1 -36020.704,E2 -36020.704} C_VEL
LIN {X 0,Y 144.136,Z 560.427,A -85,B 0,C 180,E1 -36018.65,E2 -36018.65} C_VEL
LIN {X 0,Y 153.986,Z 550.927,A -85,B 0,C 180,E1 -36017.233,E2 -36017.233} C_VEL
LIN {X 0,Y 163.115,Z 540.433,A -85,B 0,C 180,E1 -36016.116,E2 -36016.116} C_VEL
LIN {X 0,Y 171.452,Z 528.884,A -85,B 0,C 180,E1 -36015.193,E2 -36015.193} C_VEL
LIN {X 0,Y 179.074,Z 516.059,A -85,B 0,C 180,E1 -36014.538,E2 -36014.538} C_VEL
LIN {X 0,Y 185.146,Z 503.179,A -85,B 0,C 180,E1 -36014.01,E2 -36014.01} C_VEL
LIN {X 0,Y 189.923,Z 490.063,A -85,B 0,C 180,E1 -36013.596,E2 -36013.596} C_VEL
LIN {X 0,Y 190.939,Z 486.628,A -85,B 0,C 180,E1 -36013.481,E2 -36013.481} C_VEL
LIN {X 0,Y 190.921,Z 483.191,A -85,B 0,C 180,E1 -36011.117,E2 -36011.117} C_VEL
LIN {X 0,Y 190.953,Z 481.311,A -85,B 0,C 180,E1 -36009.501,E2 -36009.501} C_VEL
LIN {X 0,Y 190.989,Z 479.028,A -85,B 0,C 180,E1 -36006.317,E2 -36006.317} C_VEL
LIN {X 0,Y 190.998,Z 479.045,A -85,B 0,C 180,E1 -36003.943,E2 -36003.943} C_VEL
LIN {X 0,Y 191.051,Z 481.353,A -85,B 0,C 180,E1 -36000.263,E2 -36000.263} C_VEL
LIN {X 0,Y 191.268,Z 483.852,A -85,B 0,C 180,E1 -35997.678,E2 -35997.678} C_VEL
LIN {X 0,Y 186.994,Z 496.647,A -85,B 0,C 180,E1 -35997.109,E2 -35997.109} C_VEL
LIN {X 0,Y 181.579,Z 509.11,A -85,B 0,C 180,E1 -35996.396,E2 -35996.396} C_VEL
LIN {X 0,Y 174.643,Z 521.768,A -85,B 0,C 180,E1 -35995.497,E2 -35995.497} C_VEL
LIN {X 0,Y 167.113,Z 532.932,A -85,B 0,C 180,E1 -35994.471,E2 -35994.471} C_VEL
LIN {X 0,Y 158.702,Z 543.331,A -85,B 0,C 180,E1 -35993.184,E2 -35993.184} C_VEL
LIN {X 0,Y 148.7,Z 553.572,A -85,B 0,C 180,E1 -35991.519,E2 -35991.519} C_VEL
LIN {X 0,Y 138.809,Z 562.011,A -85,B 0,C 180,E1 -35989.688,E2 -35989.688} C_VEL
LIN {X 0,Y 128.725,Z 569.253,A -85,B 0,C 180,E1 -35987.429,E2 -35987.429} C_VEL
LIN {X 0,Y 119.623,Z 574.767,A -85,B 0,C 180,E1 -35985.014,E2 -35985.014} C_VEL
LIN {X 0,Y 110.401,Z 579.421,A -85,B 0,C 180,E1 -35982.085,E2 -35982.085} C_VEL
LIN {X 0,Y 98.597,Z 584.193,A -85,B 0,C 180,E1 -35977.42,E2 -35977.42} C_VEL
LIN {X 0,Y 87.616,Z 587.396,A -85,B 0,C 180,E1 -35971.544,E2 -35971.544} C_VEL
LIN {X 0,Y 77.75,Z 589.137,A -85,B 0,C 180,E1 -35964.151,E2 -35964.151} C_VEL
LIN {X 0,Y 69.515,Z 589.495,A -85,B 0,C 180,E1 -35954.835,E2 -35954.835} C_VEL
LIN {X 0,Y 63.266,Z 588.499,A -85,B 0,C 180,E1 -35943.593,E2 -35943.593} C_VEL
LIN {X 0,Y 59.84,Z 586.12,A -85,B 0,C 180,E1 -35930.54,E2 -35930.54} C_VEL
LIN {X 0,Y 59.196,Z 582.349,A -85,B 0,C 180,E1 -35916.779,E2 -35916.779} C_VEL
LIN {X 0,Y 61.561,Z 577.07,A -85,B 0,C 180,E1 -35903.451,E2 -35903.451} C_VEL
LIN {X 0,Y 65.016,Z 571.974,A -85,B 0,C 180,E1 -35894.36,E2 -35894.36} C_VEL
LIN {X 0,Y 70.331,Z 564.763,A -85,B 0,C 180,E1 -35884.944,E2 -35884.944} C_VEL
LIN {X 0,Y 76.109,Z 557.215,A -85,B 0,C 180,E1 -35878.035,E2 -35878.035} C_VEL
LIN {X 0,Y 82.909,Z 548.131,A -85,B 0,C 180,E1 -35872.215,E2 -35872.215} C_VEL
LIN {X 0,Y 90.376,Z 537.136,A -85,B 0,C 180,E1 -35867.286,E2 -35867.286} C_VEL
LIN {X 0,Y 96.844,Z 525.98,A -85,B 0,C 180,E1 -35863.661,E2 -35863.661} C_VEL
LIN {X 0,Y 97.29,Z 523.99,A -85,B 0,C 180,E1 -35862.641,E2 -35862.641} C_VEL
LIN {X 0,Y 95.117,Z 525.108,A -85,B 0,C 180,E1 -35861.511,E2 -35861.511} C_VEL
LIN {X 0,Y 90.83,Z 527.832,A -85,B 0,C 180,E1 -35859.526,E2 -35859.526} C_VEL
LIN {X 0,Y 86.56,Z 529.994,A -85,B 0,C 180,E1 -35856.767,E2 -35856.767} C_VEL
LIN {X 0,Y 83.896,Z 531.635,A -85,B 0,C 180,E1 -35855.07,E2 -35855.07} C_VEL
LIN {X 0,Y 74.444,Z 539.192,A -85,B 0,C 180,E1 -35850.665,E2 -35850.665} C_VEL
LIN {X 0,Y 72.061,Z 540.578,A -85,B 0,C 180,E1 -35848.461,E2 -35848.461} C_VEL
LIN {X 0,Y 69.095,Z 541.912,A -85,B 0,C 180,E1 -35843.922,E2 -35843.922} C_VEL
LIN {X 0,Y 66.789,Z 542.895,A -85,B 0,C 180,E1 -35838.338,E2 -35838.338} C_VEL
LIN {X 0,Y 63.564,Z 545.586,A -85,B 0,C 180,E1 -35826.326,E2 -35826.326} C_VEL
LIN {X 0,Y 63.882,Z 546.015,A -85,B 0,C 180,E1 -35820,E2 -35820} C_VEL
LIN {X 0,Y 64.334,Z 547.085,A -85,B 0,C 180,E1 -35813.749,E2 -35813.749} C_VEL
LIN {X 0,Y 65.573,Z 546.457,A -85,B 0,C 180,E1 -35811.94,E2 -35811.94} C_VEL
LIN {X 0,Y 65.952,Z 546.294,A -85,B 0,C 180,E1 -35811.603,E2 -35811.603} C_VEL
LIN {X 0,Y 67.757,Z 554.326,A -85,B 0,C 180,E1 -35805.022,E2 -35805.022} C_VEL
LIN {X 0,Y 71.899,Z 564.778,A -85,B 0,C 180,E1 -35795.422,E2 -35795.422} C_VEL
LIN {X 0,Y 78.755,Z 574.724,A -85,B 0,C 180,E1 -35786.229,E2 -35786.229} C_VEL
LIN {X 0,Y 84.094,Z 580.251,A -85,B 0,C 180,E1 -35781.409,E2 -35781.409} C_VEL
LIN {X 0,Y 82.85,Z 579.168,A -85,B 0,C 180,E1 -35779.56,E2 -35779.56} C_VEL
LIN {X 0,Y 74.603,Z 569.579,A -85,B 0,C 180,E1 -35769.821,E2 -35769.821} C_VEL
LIN {X 0,Y 74.161,Z 569.002,A -85,B 0,C 180,E1 -35769.149,E2 -35769.149} C_VEL
LIN {X 0,Y 67.073,Z 574.91,A -85,B 0,C 180,E1 -35763.795,E2 -35763.795} C_VEL
LIN {X 0,Y 61.611,Z 579.83,A -85,B 0,C 180,E1 -35757.067,E2 -35757.067} C_VEL
LIN {X 0,Y 55.899,Z 585.898,A -85,B 0,C 180,E1 -35744.531,E2 -35744.531} C_VEL
LIN {X 0,Y 53.264,Z 589.317,A -85,B 0,C 180,E1 -35733.788,E2 -35733.788} C_VEL
LIN {X 0,Y 52.259,Z 591.939,A -85,B 0,C 180,E1 -35722.316,E2 -35722.316} C_VEL
LIN {X 0,Y 54.289,Z 594.21,A -85,B 0,C 180,E1 -35707.248,E2 -35707.248} C_VEL
LIN {X 0,Y 59.714,Z 595.19,A -85,B 0,C 180,E1 -35694.112,E2 -35694.112} C_VEL
LIN {X 0,Y 67.718,Z 594.895,A -85,B 0,C 180,E1 -35683.633,E2 -35683.633} C_VEL
LIN {X 0,Y 77.466,Z 593.321,A -85,B 0,C 180,E1 -35675.557,E2 -35675.557} C_VEL
LIN {X 0,Y 88.503,Z 590.443,A -85,B 0,C 180,E1 -35669.499,E2 -35669.499} C_VEL
LIN {X 0,Y 100.385,Z 586.177,A -85,B 0,C 180,E1 -35664.92,E2 -35664.92} C_VEL
LIN {X 0,Y 112.834,Z 580.396,A -85,B 0,C 180,E1 -35661.41,E2 -35661.41} C_VEL
LIN {X 0,Y 124.053,Z 573.937,A -85,B 0,C 180,E1 -35658.985,E2 -35658.985} C_VEL
LIN {X 0,Y 135.449,Z 565.961,A -85,B 0,C 180,E1 -35656.953,E2 -35656.953} C_VEL
LIN {X 0,Y 145.36,Z 557.659,A -85,B 0,C 180,E1 -35655.506,E2 -35655.506} C_VEL
LIN {X 0,Y 155.409,Z 547.692,A -85,B 0,C 180,E1 -35654.327,E2 -35654.327} C_VEL
LIN {X 0,Y 164.661,Z 536.643,A -85,B 0,C 180,E1 -35653.357,E2 -35653.357} C_VEL
LIN {X 0,Y 173.142,Z 524.308,A -85,B 0,C 180,E1 -35652.614,E2 -35652.614} C_VEL
LIN {X 0,Y 180.527,Z 510.988,A -85,B 0,C 180,E1 -35652.098,E2 -35652.098} C_VEL
LIN {X 0,Y 186.562,Z 496.967,A -85,B 0,C 180,E1 -35651.635,E2 -35651.635} C_VEL
LIN {X 0,Y 188.087,Z 492.704,A -85,B 0,C 180,E1 -35651.524,E2 -35651.524} C_VEL
LIN {X 0,Y 188.684,Z 490.764,A -85,B 0,C 180,E1 -35651.363,E2 -35651.363} C_VEL
LIN {X 0,Y 188.848,Z 488.577,A -85,B 0,C 180,E1 -35649.608,E2 -35649.608} C_VEL
LIN {X 0,Y 189.06,Z 486.001,A -85,B 0,C 180,E1 -35646.381,E2 -35646.381} C_VEL
LIN {X 0,Y 189.082,Z 485.802,A -85,B 0,C 180,E1 -35644.249,E2 -35644.249} C_VEL
LIN {X 0,Y 188.946,Z 487.02,A -85,B 0,C 180,E1 -35642.125,E2 -35642.125} C_VEL
LIN {X 0,Y 188.886,Z 488.909,A -85,B 0,C 180,E1 -35639.69,E2 -35639.69} C_VEL
LIN {X 0,Y 188.587,Z 489.918,A -85,B 0,C 180,E1 -35639.551,E2 -35639.551} C_VEL
LIN {X 0,Y 183.487,Z 503.138,A -85,B 0,C 180,E1 -35638.983,E2 -35638.983} C_VEL
LIN {X 0,Y 176.931,Z 516.341,A -85,B 0,C 180,E1 -35638.184,E2 -35638.184} C_VEL
LIN {X 0,Y 169.221,Z 528.635,A -85,B 0,C 180,E1 -35637.302,E2 -35637.302} C_VEL
LIN {X 0,Y 161.421,Z 538.927,A -85,B 0,C 180,E1 -35636.288,E2 -35636.288} C_VEL
LIN {X 0,Y 151.263,Z 549.982,A -85,B 0,C 180,E1 -35634.857,E2 -35634.857} C_VEL
LIN {X 0,Y 141.046,Z 559.18,A -85,B 0,C 180,E1 -35633.255,E2 -35633.255} C_VEL
LIN {X 0,Y 131.039,Z 566.728,A -85,B 0,C 180,E1 -35631.392,E2 -35631.392} C_VEL
LIN {X 0,Y 121.19,Z 572.971,A -85,B 0,C 180,E1 -35629.234,E2 -35629.234} C_VEL
LIN {X 0,Y 111.534,Z 578.09,A -85,B 0,C 180,E1 -35626.716,E2 -35626.716} C_VEL
LIN {X 0,Y 99.066,Z 583.324,A -85,B 0,C 180,E1 -35622.616,E2 -35622.616} C_VEL
LIN {X 0,Y 90.089,Z 586.217,A -85,B 0,C 180,E1 -35618.875,E2 -35618.875} C_VEL
LIN {X 0,Y 78.895,Z 588.773,A -85,B 0,C 180,E1 -35612.572,E2 -35612.572} C_VEL
LIN {X 0,Y 68.893,Z 589.896,A -85,B 0,C 180,E1 -35604.401,E2 -35604.401} C_VEL
LIN {X 0,Y 60.643,Z 589.645,A -85,B 0,C 180,E1 -35593.847,E2 -35593.847} C_VEL
LIN {X 0,Y 54.768,Z 588.035,A -85,B 0,C 180,E1 -35580.748,E2 -35580.748} C_VEL
LIN {X 0,Y 52.889,Z 586.45,A -85,B 0,C 180,E1 -35572.02,E2 -35572.02} C_VEL
LIN {X 0,Y 52.035,Z 583.003,A -85,B 0,C 180,E1 -35557.717,E2 -35557.717} C_VEL
LIN {X 0,Y 54.447,Z 577.799,A -85,B 0,C 180,E1 -35542.591,E2 -35542.591} C_VEL
LIN {X 0,Y 58.183,Z 572.782,A -85,B 0,C 180,E1 -35532.467,E2 -35532.467} C_VEL
LIN {X 0,Y 63.97,Z 565.66,A -85,B 0,C 180,E1 -35522.25,E2 -35522.25} C_VEL
LIN {X 0,Y 70.159,Z 558.221,A -85,B 0,C 180,E1 -35514.95,E2 -35514.95} C_VEL
LIN {X 0,Y 77.435,Z 549.247,A -85,B 0,C 180,E1 -35509.004,E2 -35509.004} C_VEL
LIN {X 0,Y 83.942,Z 540.35,A -85,B 0,C 180,E1 -35504.809,E2 -35504.809} C_VEL
LIN {X 0,Y 87.61,Z 534.928,A -85,B 0,C 180,E1 -35502.859,E2 -35502.859} C_VEL
LIN {X 0,Y 88.29,Z 533.382,A -85,B 0,C 180,E1 -35502.033,E2 -35502.033} C_VEL
LIN {X 0,Y 76.401,Z 538.716,A -85,B 0,C 180,E1 -35493.372,E2 -35493.372} C_VEL
LIN {X 0,Y 72.061,Z 540.578,A -85,B 0,C 180,E1 -35488.461,E2 -35488.461} C_VEL
LIN {X 0,Y 69.86,Z 541.847,A -85,B 0,C 180,E1 -35485.967,E2 -35485.967} C_VEL
LIN {X 0,Y 61.873,Z 547.977,A -85,B 0,C 180,E1 -35478.178,E2 -35478.178} C_VEL
LIN {X 0,Y 60.274,Z 549.143,A -85,B 0,C 180,E1 -35474.951,E2 -35474.951} C_VEL
LIN {X 0,Y 58.579,Z 550.597,A -85,B 0,C 180,E1 -35466.867,E2 -35466.867} C_VEL
LIN {X 0,Y 58.831,Z 551.055,A -85,B 0,C 180,E1 -35460,E2 -35460} C_VEL
LIN {X 0,Y 59.551,Z 552.506,A -85,B 0,C 180,E1 -35450.963,E2 -35450.963} C_VEL
LIN {X 0,Y 60.262,Z 553.405,A -85,B 0,C 180,E1 -35446.557,E2 -35446.557} C_VEL
LIN {X 0,Y 62.415,Z 554.333,A -85,B 0,C 180,E1 -35440.325,E2 -35440.325} C_VEL
LIN {X 0,Y 64.186,Z 553.945,A -85,B 0,C 180,E1 -35438.599,E2 -35438.599} C_VEL
LIN {X 0,Y 69.102,Z 563.597,A -85,B 0,C 180,E1 -35429.547,E2 -35429.547} C_VEL
LIN {X 0,Y 76.337,Z 572.781,A -85,B 0,C 180,E1 -35421.278,E2 -35421.278} C_VEL
LIN {X 0,Y 75.334,Z 571.751,A -85,B 0,C 180,E1 -35419.394,E2 -35419.394} C_VEL
LIN {X 0,Y 70.926,Z 566.482,A -85,B 0,C 180,E1 -35413.964,E2 -35413.964} C_VEL
LIN {X 0,Y 63.116,Z 572.601,A -85,B 0,C 180,E1 -35409.027,E2 -35409.027} C_VEL
LIN {X 0,Y 55.421,Z 579.045,A -85,B 0,C 180,E1 -35400.388,E2 -35400.388} C_VEL
LIN {X 0,Y 49.102,Z 585.193,A -85,B 0,C 180,E1 -35386.597,E2 -35386.597} C_VEL
LIN {X 0,Y 46.2,Z 588.684,A -85,B 0,C 180,E1 -35374.369,E2 -35374.369} C_VEL
LIN {X 0,Y 45.221,Z 591.361,A -85,B 0,C 180,E1 -35361.111,E2 -35361.111} C_VEL
LIN {X 0,Y 47.803,Z 593.709,A -85,B 0,C 180,E1 -35343.946,E2 -35343.946} C_VEL
LIN {X 0,Y 54.105,Z 594.758,A -85,B 0,C 180,E1 -35329.686,E2 -35329.686} C_VEL
LIN {X 0,Y 63.017,Z 594.53,A -85,B 0,C 180,E1 -35318.942,E2 -35318.942} C_VEL
LIN {X 0,Y 73.554,Z 593.023,A -85,B 0,C 180,E1 -35311.039,E2 -35311.039} C_VEL
LIN {X 0,Y 85.224,Z 590.214,A -85,B 0,C 180,E1 -35305.33,E2 -35305.33} C_VEL
LIN {X 0,Y 97.6,Z 586.02,A -85,B 0,C 180,E1 -35301.128,E2 -35301.128} C_VEL
LIN {X 0,Y 110.435,Z 580.316,A -85,B 0,C 180,E1 -35297.97,E2 -35297.97} C_VEL
LIN {X 0,Y 123.58,Z 572.928,A -85,B 0,C 180,E1 -35295.55,E2 -35295.55} C_VEL
LIN {X 0,Y 135.225,Z 564.824,A -85,B 0,C 180,E1 -35293.813,E2 -35293.813} C_VEL
LIN {X 0,Y 145.317,Z 556.376,A -85,B 0,C 180,E1 -35292.594,E2 -35292.594} C_VEL
LIN {X 0,Y 155.503,Z 546.226,A -85,B 0,C 180,E1 -35291.599,E2 -35291.599} C_VEL
LIN {X 0,Y 164.866,Z 534.899,A -85,B 0,C 180,E1 -35290.778,E2 -35290.778} C_VEL
LIN {X 0,Y 172.597,Z 523.654,A -85,B 0,C 180,E1 -35290.259,E2 -35290.259} C_VEL
LIN {X 0,Y 179.667,Z 511.041,A -85,B 0,C 180,E1 -35289.857,E2 -35289.857} C_VEL
LIN {X 0,Y 185.586,Z 497.596,A -85,B 0,C 180,E1 -35289.481,E2 -35289.481} C_VEL
LIN {X 0,Y 186.092,Z 496.271,A -85,B 0,C 180,E1 -35289.444,E2 -35289.444} C_VEL
LIN {X 0,Y 186.453,Z 495.132,A -85,B 0,C 180,E1 -35289.133,E2 -35289.133} C_VEL
LIN {X 0,Y 186.81,Z 492.856,A -85,B 0,C 180,E1 -35286.459,E2 -35286.459} C_VEL
LIN {X 0,Y 186.83,Z 492.605,A -85,B 0,C 180,E1 -35284.3,E2 -35284.3} C_VEL
LIN {X 0,Y 186.511,Z 494.258,A -85,B 0,C 180,E1 -35281.614,E2 -35281.614} C_VEL
LIN {X 0,Y 180.942,Z 507.426,A -85,B 0,C 180,E1 -35280.985,E2 -35280.985} C_VEL
LIN {X 0,Y 173.835,Z 520.527,A -85,B 0,C 180,E1 -35280.248,E2 -35280.248} C_VEL
LIN {X 0,Y 166.342,Z 531.69,A -85,B 0,C 180,E1 -35279.486,E2 -35279.486} C_VEL
LIN {X 0,Y 157.638,Z 542.45,A -85,B 0,C 180,E1 -35278.456,E2 -35278.456} C_VEL
LIN {X 0,Y 147.256,Z 553.053,A -85,B 0,C 180,E1 -35277.147,E2 -35277.147} C_VEL
LIN {X 0,Y 136.954,Z 561.74,A -85,B 0,C 180,E1 -35275.691,E2 -35275.691} C_VEL
LIN {X 0,Y 126.761,Z 568.906,A -85,B 0,C 180,E1 -35273.974,E2 -35273.974} C_VEL
LIN {X 0,Y 116.703,Z 574.81,A -85,B 0,C 180,E1 -35271.956,E2 -35271.956} C_VEL
LIN {X 0,Y 106.81,Z 579.637,A -85,B 0,C 180,E1 -35269.578,E2 -35269.578} C_VEL
LIN {X 0,Y 93.959,Z 584.569,A -85,B 0,C 180,E1 -35265.68,E2 -35265.68} C_VEL
LIN {X 0,Y 81.651,Z 587.944,A -85,B 0,C 180,E1 -35260.633,E2 -35260.633} C_VEL
LIN {X 0,Y 70.182,Z 589.869,A -85,B 0,C 180,E1 -35253.893,E2 -35253.893} C_VEL
LIN {X 0,Y 60.035,Z 590.383,A -85,B 0,C 180,E1 -35244.727,E2 -35244.727} C_VEL
LIN {X 0,Y 51.754,Z 589.527,A -85,B 0,C 180,E1 -35232.561,E2 -35232.561} C_VEL
LIN {X 0,Y 46.485,Z 587.29,A -85,B 0,C 180,E1 -35216.851,E2 -35216.851} C_VEL
LIN {X 0,Y 44.907,Z 583.657,A -85,B 0,C 180,E1 -35198.951,E2 -35198.951} C_VEL
LIN {X 0,Y 47.335,Z 578.529,A -85,B 0,C 180,E1 -35181.47,E2 -35181.47} C_VEL
LIN {X 0,Y 51.406,Z 573.594,A -85,B 0,C 180,E1 -35170.064,E2 -35170.064} C_VEL
LIN {X 0,Y 57.783,Z 566.557,A -85,B 0,C 180,E1 -35158.971,E2 -35158.971} C_VEL
LIN {X 0,Y 64.46,Z 559.224,A -85,B 0,C 180,E1 -35151.313,E2 -35151.313} C_VEL
LIN {X 0,Y 72.217,Z 550.369,A -85,B 0,C 180,E1 -35145.298,E2 -35145.298} C_VEL
LIN {X 0,Y 78.356,Z 542.596,A -85,B 0,C 180,E1 -35141.51,E2 -35141.51} C_VEL
LIN {X 0,Y 78.113,Z 541.777,A -85,B 0,C 180,E1 -35140.192,E2 -35140.192} C_VEL
LIN {X 0,Y 68.565,Z 545.5,A -85,B 0,C 180,E1 -35131.447,E2 -35131.447} C_VEL
LIN {X 0,Y 64.638,Z 547.041,A -85,B 0,C 180,E1 -35125.687,E2 -35125.687} C_VEL
LIN {X 0,Y 62.073,Z 548.054,A -85,B 0,C 180,E1 -35119.787,E2 -35119.787} C_VEL
LIN {X 0,Y 60.274,Z 549.143,A -85,B 0,C 180,E1 -35114.951,E2 -35114.951} C_VEL
LIN {X 0,Y 57.831,Z 551.268,A -85,B 0,C 180,E1 -35107.904,E2 -35107.904} C_VEL
LIN {X 0,Y 54.334,Z 556.511,A -85,B 0,C 180,E1 -35092.893,E2 -35092.893} C_VEL
LIN {X 0,Y 54.727,Z 557.864,A -85,B 0,C 180,E1 -35086.861,E2 -35086.861} C_VEL
LIN {X 0,Y 55.188,Z 558.157,A -85,B 0,C 180,E1 -35084.888,E2 -35084.888} C_VEL
LIN {X 0,Y 57.413,Z 558.992,A -85,B 0,C 180,E1 -35078.531,E2 -35078.531} C_VEL
LIN {X 0,Y 59.821,Z 560.491,A -85,B 0,C 180,E1 -35072.072,E2 -35072.072} C_VEL
LIN {X 0,Y 63.242,Z 561.662,A -85,B 0,C 180,E1 -35066.373,E2 -35066.373} C_VEL
LIN {X 0,Y 66.427,Z 561.409,A -85,B 0,C 180,E1 -35064.087,E2 -35064.087} C_VEL
LIN {X 0,Y 69.015,Z 564.756,A -85,B 0,C 180,E1 -35061.098,E2 -35061.098} C_VEL
LIN {X 0,Y 68.35,Z 563.94,A -85,B 0,C 180,E1 -35059.259,E2 -35059.259} C_VEL
LIN {X 0,Y 68.017,Z 563.943,A -85,B 0,C 180,E1 -35059.08,E2 -35059.08} C_VEL
LIN {X 0,Y 59.69,Z 570.334,A -85,B 0,C 180,E1 -35054.777,E2 -35054.777} C_VEL
LIN {X 0,Y 51.708,Z 576.453,A -85,B 0,C 180,E1 -35047.582,E2 -35047.582} C_VEL
LIN {X 0,Y 45.483,Z 581.58,A -85,B 0,C 180,E1 -35037.54,E2 -35037.54} C_VEL
LIN {X 0,Y 41.137,Z 585.79,A -85,B 0,C 180,E1 -35024.822,E2 -35024.822} C_VEL
LIN {X 0,Y 38.553,Z 589.05,A -85,B 0,C 180,E1 -35010.025,E2 -35010.025} C_VEL
LIN {X 0,Y 39.308,Z 592.145,A -85,B 0,C 180,E1 -34989.149,E2 -34989.149} C_VEL
LIN {X 0,Y 44.809,Z 593.911,A -85,B 0,C 180,E1 -34971.326,E2 -34971.326} C_VEL
LIN {X 0,Y 53.601,Z 594.391,A -85,B 0,C 180,E1 -34958.396,E2 -34958.396} C_VEL
LIN {X 0,Y 64.314,Z 593.595,A -85,B 0,C 180,E1 -34949.425,E2 -34949.425} C_VEL
LIN {X 0,Y 76.214,Z 591.52,A -85,B 0,C 180,E1 -34943.247,E2 -34943.247} C_VEL
LIN {X 0,Y 88.81,Z 588.105,A -85,B 0,C 180,E1 -34938.874,E2 -34938.874} C_VEL
LIN {X 0,Y 101.828,Z 583.247,A -85,B 0,C 180,E1 -34935.671,E2 -34935.671} C_VEL
LIN {X 0,Y 115.146,Z 576.808,A -85,B 0,C 180,E1 -34933.311,E2 -34933.311} C_VEL
LIN {X 0,Y 126.931,Z 569.692,A -85,B 0,C 180,E1 -34931.665,E2 -34931.665} C_VEL
LIN {X 0,Y 138.808,Z 560.934,A -85,B 0,C 180,E1 -34930.309,E2 -34930.309} C_VEL
LIN {X 0,Y 149.074,Z 551.806,A -85,B 0,C 180,E1 -34929.397,E2 -34929.397} C_VEL
LIN {X 0,Y 159.398,Z 540.775,A -85,B 0,C 180,E1 -34928.661,E2 -34928.661} C_VEL
LIN {X 0,Y 168.014,Z 529.564,A -85,B 0,C 180,E1 -34928.106,E2 -34928.106} C_VEL
LIN {X 0,Y 175.822,Z 517.175,A -85,B 0,C 180,E1 -34927.751,E2 -34927.751} C_VEL
LIN {X 0,Y 181.965,Z 505.104,A -85,B 0,C 180,E1 -34927.471,E2 -34927.471} C_VEL
LIN {X 0,Y 183.612,Z 501.338,A -85,B 0,C 180,E1 -34927.368,E2 -34927.368} C_VEL
LIN {X 0,Y 184.183,Z 499.742,A -85,B 0,C 180,E1 -34926.551,E2 -34926.551} C_VEL
LIN {X 0,Y 184.26,Z 499.295,A -85,B 0,C 180,E1 -34924.36,E2 -34924.36} C_VEL
LIN {X 0,Y 184.128,Z 499.689,A -85,B 0,C 180,E1 -34923.66,E2 -34923.66} C_VEL
LIN {X 0,Y 179.209,Z 510.337,A -85,B 0,C 180,E1 -34923.115,E2 -34923.115} C_VEL
LIN {X 0,Y 172.007,Z 522.976,A -85,B 0,C 180,E1 -34922.477,E2 -34922.477} C_VEL
LIN {X 0,Y 163.784,Z 534.627,A -85,B 0,C 180,E1 -34921.731,E2 -34921.731} C_VEL
LIN {X 0,Y 154.091,Z 545.848,A -85,B 0,C 180,E1 -34920.739,E2 -34920.739} C_VEL
LIN {X 0,Y 143.507,Z 555.928,A -85,B 0,C 180,E1 -34919.56,E2 -34919.56} C_VEL
LIN {X 0,Y 133.125,Z 564.128,A -85,B 0,C 180,E1 -34918.281,E2 -34918.281} C_VEL
LIN {X 0,Y 121.624,Z 571.634,A -85,B 0,C 180,E1 -34916.55,E2 -34916.55} C_VEL
LIN {X 0,Y 109.105,Z 578.224,A -85,B 0,C 180,E1 -34914.216,E2 -34914.216} C_VEL
LIN {X 0,Y 95.657,Z 583.711,A -85,B 0,C 180,E1 -34910.991,E2 -34910.991} C_VEL
LIN {X 0,Y 85.908,Z 586.67,A -85,B 0,C 180,E1 -34908.014,E2 -34908.014} C_VEL
LIN {X 0,Y 73.308,Z 589.383,A -85,B 0,C 180,E1 -34902.792,E2 -34902.792} C_VEL
LIN {X 0,Y 61.536,Z 590.681,A -85,B 0,C 180,E1 -34895.55,E2 -34895.55} C_VEL
LIN {X 0,Y 51.12,Z 590.598,A -85,B 0,C 180,E1 -34885.263,E2 -34885.263} C_VEL
LIN {X 0,Y 42.913,Z 589.133,A -85,B 0,C 180,E1 -34870.729,E2 -34870.729} C_VEL
LIN {X 0,Y 38.395,Z 586.271,A -85,B 0,C 180,E1 -34851.372,E2 -34851.372} C_VEL
LIN {X 0,Y 38.409,Z 581.983,A -85,B 0,C 180,E1 -34829.975,E2 -34829.975} C_VEL
LIN {X 0,Y 41.557,Z 577.767,A -85,B 0,C 180,E1 -34815.331,E2 -34815.331} C_VEL
LIN {X 0,Y 47.731,Z 571.491,A -85,B 0,C 180,E1 -34801.194,E2 -34801.194} C_VEL
LIN {X 0,Y 55.326,Z 564.006,A -85,B 0,C 180,E1 -34790.705,E2 -34790.705} C_VEL
LIN {X 0,Y 63.186,Z 556.051,A -85,B 0,C 180,E1 -34783.879,E2 -34783.879} C_VEL
LIN {X 0,Y 67.952,Z 550.798,A -85,B 0,C 180,E1 -34780.667,E2 -34780.667} C_VEL
LIN {X 0,Y 68.972,Z 548.903,A -85,B 0,C 180,E1 -34778.732,E2 -34778.732} C_VEL
LIN {X 0,Y 60.04,Z 551.934,A -85,B 0,C 180,E1 -34767.817,E2 -34767.817} C_VEL
LIN {X 0,Y 55.576,Z 553.795,A -85,B 0,C 180,E1 -34757.412,E2 -34757.412} C_VEL
LIN {X 0,Y 53.365,Z 555.368,A -85,B 0,C 180,E1 -34747.542,E2 -34747.542} C_VEL
LIN {X 0,Y 53.56,Z 555.834,A -85,B 0,C 180,E1 -34740,E2 -34740} C_VEL
LIN {X 0,Y 55.188,Z 558.157,A -85,B 0,C 180,E1 -34724.888,E2 -34724.888} C_VEL
LIN {X 0,Y 55.804,Z 559.154,A -85,B 0,C 180,E1 -34720.971,E2 -34720.971} C_VEL
LIN {X 0,Y 55.671,Z 561.931,A -85,B 0,C 180,E1 -34714.634,E2 -34714.634} C_VEL
LIN {X 0,Y 56.125,Z 564.661,A -85,B 0,C 180,E1 -34708.297,E2 -34708.297} C_VEL
LIN {X 0,Y 57.654,Z 565.679,A -85,B 0,C 180,E1 -34704.732,E2 -34704.732} C_VEL
LIN {X 0,Y 58.636,Z 565.947,A -85,B 0,C 180,E1 -34703.324,E2 -34703.324} C_VEL
LIN {X 0,Y 57.853,Z 567.242,A -85,B 0,C 180,E1 -34701.591,E2 -34701.591} C_VEL
LIN {X 0,Y 49.036,Z 573.687,A -85,B 0,C 180,E1 -34695.606,E2 -34695.606} C_VEL
LIN {X 0,Y 41.558,Z 579.239,A -85,B 0,C 180,E1 -34686.179,E2 -34686.179} C_VEL
LIN {X 0,Y 35.818,Z 583.784,A -85,B 0,C 180,E1 -34673.053,E2 -34673.053} C_VEL
LIN {X 0,Y 32.083,Z 587.417,A -85,B 0,C 180,E1 -34656.297,E2 -34656.297} C_VEL
LIN {X 0,Y 31.253,Z 590.163,A -85,B 0,C 180,E1 -34637.081,E2 -34637.081} C_VEL
LIN {X 0,Y 35.577,Z 592.657,A -85,B 0,C 180,E1 -34613.832,E2 -34613.832} C_VEL
LIN {X 0,Y 44.206,Z 593.845,A -85,B 0,C 180,E1 -34597.642,E2 -34597.642} C_VEL
LIN {X 0,Y 55.167,Z 593.757,A -85,B 0,C 180,E1 -34587.32,E2 -34587.32} C_VEL
LIN {X 0,Y 67.332,Z 592.397,A -85,B 0,C 180,E1 -34580.613,E2 -34580.613} C_VEL
LIN {X 0,Y 80.177,Z 589.743,A -85,B 0,C 180,E1 -34576.105,E2 -34576.105} C_VEL
LIN {X 0,Y 93.415,Z 585.706,A -85,B 0,C 180,E1 -34572.95,E2 -34572.95} C_VEL
LIN {X 0,Y 106.911,Z 580.157,A -85,B 0,C 180,E1 -34570.713,E2 -34570.713} C_VEL
LIN {X 0,Y 120.555,Z 572.935,A -85,B 0,C 180,E1 -34569.043,E2 -34569.043} C_VEL
LIN {X 0,Y 132.555,Z 565.017,A -85,B 0,C 180,E1 -34567.847,E2 -34567.847} C_VEL
LIN {X 0,Y 142.899,Z 556.778,A -85,B 0,C 180,E1 -34567.044,E2 -34567.044} C_VEL
LIN {X 0,Y 153.286,Z 546.887,A -85,B 0,C 180,E1 -34566.411,E2 -34566.411} C_VEL
LIN {X 0,Y 162.814,Z 535.933,A -85,B 0,C 180,E1 -34565.879,E2 -34565.879} C_VEL
LIN {X 0,Y 171.519,Z 523.761,A -85,B 0,C 180,E1 -34565.554,E2 -34565.554} C_VEL
LIN {X 0,Y 175.88,Z 516.496,A -85,B 0,C 180,E1 -34565.428,E2 -34565.428} C_VEL
LIN {X 0,Y 175.797,Z 516.61,A -85,B 0,C 180,E1 -34565.137,E2 -34565.137} C_VEL
LIN {X 0,Y 167.74,Z 529.238,A -85,B 0,C 180,E1 -34564.552,E2 -34564.552} C_VEL
LIN {X 0,Y 158.81,Z 540.569,A -85,B 0,C 180,E1 -34563.826,E2 -34563.826} C_VEL
LIN {X 0,Y 149.026,Z 550.805,A -85,B 0,C 180,E1 -34562.98,E2 -34562.98} C_VEL
LIN {X 0,Y 138.401,Z 560.015,A -85,B 0,C 180,E1 -34561.978,E2 -34561.978} C_VEL
LIN {X 0,Y 126.068,Z 568.762,A -85,B 0,C 180,E1 -34560.593,E2 -34560.593} C_VEL
LIN {X 0,Y 115.567,Z 574.855,A -85,B 0,C 180,E1 -34559.157,E2 -34559.157} C_VEL
LIN {X 0,Y 105.152,Z 579.854,A -85,B 0,C 180,E1 -34557.449,E2 -34557.449} C_VEL
LIN {X 0,Y 91.446,Z 584.946,A -85,B 0,C 180,E1 -34554.593,E2 -34554.593} C_VEL
LIN {X 0,Y 78.03,Z 588.472,A -85,B 0,C 180,E1 -34550.822,E2 -34550.822} C_VEL
LIN {X 0,Y 65.087,Z 590.543,A -85,B 0,C 180,E1 -34545.53,E2 -34545.53} C_VEL
LIN {X 0,Y 52.951,Z 591.22,A -85,B 0,C 180,E1 -34537.764,E2 -34537.764} C_VEL
LIN {X 0,Y 42.194,Z 590.535,A -85,B 0,C 180,E1 -34526.058,E2 -34526.058} C_VEL
LIN {X 0,Y 34.122,Z 588.463,A -85,B 0,C 180,E1 -34507.975,E2 -34507.975} C_VEL
LIN {X 0,Y 31.77,Z 586.889,A -85,B 0,C 180,E1 -34496.13,E2 -34496.13} C_VEL
LIN {X 0,Y 31.207,Z 582.676,A -85,B 0,C 180,E1 -34469.969,E2 -34469.969} C_VEL
LIN {X 0,Y 34.668,Z 578.531,A -85,B 0,C 180,E1 -34452.329,E2 -34452.329} C_VEL
LIN {X 0,Y 40.376,Z 573.391,A -85,B 0,C 180,E1 -34438.61,E2 -34438.61} C_VEL
LIN {X 0,Y 48.744,Z 566.12,A -85,B 0,C 180,E1 -34426.929,E2 -34426.929} C_VEL
LIN {X 0,Y 56.968,Z 558.513,A -85,B 0,C 180,E1 -34419.759,E2 -34419.759} C_VEL
LIN {X 0,Y 59.499,Z 556.092,A -85,B 0,C 180,E1 -34418.228,E2 -34418.228} C_VEL
LIN {X 0,Y 59.366,Z 555.359,A -85,B 0,C 180,E1 -34416.152,E2 -34416.152} C_VEL
LIN {X 0,Y 47.948,Z 559.881,A -85,B 0,C 180,E1 -34388.4,E2 -34388.4} C_VEL
LIN {X 0,Y 48.062,Z 560.364,A -85,B 0,C 180,E1 -34380,E2 -34380} C_VEL
LIN {X 0,Y 52.177,Z 563.483,A -85,B 0,C 180,E1 -34356.25,E2 -34356.25} C_VEL
LIN {X 0,Y 54.897,Z 564.865,A -85,B 0,C 180,E1 -34349.311,E2 -34349.311} C_VEL
LIN {X 0,Y 57.654,Z 565.679,A -85,B 0,C 180,E1 -34344.732,E2 -34344.732} C_VEL
LIN {X 0,Y 57.72,Z 566.23,A -85,B 0,C 180,E1 -34343.624,E2 -34343.624} C_VEL
LIN {X 0,Y 56.352,Z 567.616,A -85,B 0,C 180,E1 -34342.217,E2 -34342.217} C_VEL
LIN {X 0,Y 53.298,Z 569.539,A -85,B 0,C 180,E1 -34341.193,E2 -34341.193} C_VEL
LIN {X 0,Y 44.111,Z 573.61,A -85,B 0,C 180,E1 -34340.281,E2 -34340.281} C_VEL
LIN {X 0,Y 40.494,Z 575.497,A -85,B 0,C 180,E1 -34338.448,E2 -34338.448} C_VEL
LIN {X 0,Y 39.875,Z 575.876,A -85,B 0,C 180,E1 -34337.825,E2 -34337.825} C_VEL
LIN {X 0,Y 31.424,Z 581.663,A -85,B 0,C 180,E1 -34323.903,E2 -34323.903} C_VEL
LIN {X 0,Y 26.2,Z 585.63,A -85,B 0,C 180,E1 -34305.545,E2 -34305.545} C_VEL
LIN {X 0,Y 24.384,Z 589.564,A -85,B 0,C 180,E1 -34273.349,E2 -34273.349} C_VEL
LIN {X 0,Y 30.133,Z 592.126,A -85,B 0,C 180,E1 -34245.831,E2 -34245.831} C_VEL
LIN {X 0,Y 40.253,Z 593.379,A -85,B 0,C 180,E1 -34229.586,E2 -34229.586} C_VEL
LIN {X 0,Y 52.279,Z 593.357,A -85,B 0,C 180,E1 -34220.359,E2 -34220.359} C_VEL
LIN {X 0,Y 65.164,Z 592.064,A -85,B 0,C 180,E1 -34214.73,E2 -34214.73} C_VEL
LIN {X 0,Y 78.503,Z 589.481,A -85,B 0,C 180,E1 -34211.115,E2 -34211.115} C_VEL
LIN {X 0,Y 92.082,Z 585.535,A -85,B 0,C 180,E1 -34208.633,E2 -34208.633} C_VEL
LIN {X 0,Y 105.822,Z 580.077,A -85,B 0,C 180,E1 -34206.935,E2 -34206.935} C_VEL
LIN {X 0,Y 119.643,Z 572.939,A -85,B 0,C 180,E1 -34205.677,E2 -34205.677} C_VEL
LIN {X 0,Y 131.775,Z 565.113,A -85,B 0,C 180,E1 -34204.792,E2 -34204.792} C_VEL
LIN {X 0,Y 133.511,Z 563.879,A -85,B 0,C 180,E1 -34204.686,E2 -34204.686} C_VEL
LIN {X 0,Y 133.485,Z 563.884,A -85,B 0,C 180,E1 -34204.544,E2 -34204.544} C_VEL
LIN {X 0,Y 121.082,Z 571.895,A -85,B 0,C 180,E1 -34203.366,E2 -34203.366} C_VEL
LIN {X 0,Y 108.611,Z 578.356,A -85,B 0,C 180,E1 -34201.916,E2 -34201.916} C_VEL
LIN {X 0,Y 95.656,Z 583.597,A -85,B 0,C 180,E1 -34200,E2 -34200} C_VEL
LIN {X 0,Y 84.096,Z 587.124,A -85,B 0,C 180,E1 -34197.812,E2 -34197.812} C_VEL
LIN {X 0,Y 70.38,Z 589.985,A -85,B 0,C 180,E1 -34194.256,E2 -34194.256} C_VEL
LIN {X 0,Y 57.055,Z 591.427,A -85,B 0,C 180,E1 -34189.056,E2 -34189.056} C_VEL
LIN {X 0,Y 44.448,Z 591.491,A -85,B 0,C 180,E1 -34180.931,E2 -34180.931} C_VEL
LIN {X 0,Y 33.259,Z 590.197,A -85,B 0,C 180,E1 -34167.339,E2 -34167.339} C_VEL
LIN {X 0,Y 25.461,Z 587.506,A -85,B 0,C 180,E1 -34143.335,E2 -34143.335} C_VEL
LIN {X 0,Y 24.012,Z 583.368,A -85,B 0,C 180,E1 -34109.959,E2 -34109.959} C_VEL
LIN {X 0,Y 27.899,Z 579.269,A -85,B 0,C 180,E1 -34087.84,E2 -34087.84} C_VEL
LIN {X 0,Y 34.496,Z 574.2,A -85,B 0,C 180,E1 -34072.437,E2 -34072.437} C_VEL
LIN {X 0,Y 43.503,Z 567.273,A -85,B 0,C 180,E1 -34060.894,E2 -34060.894} C_VEL
LIN {X 0,Y 51.165,Z 560.873,A -85,B 0,C 180,E1 -34054.744,E2 -34054.744} C_VEL
LIN {X 0,Y 42.355,Z 564.119,A -85,B 0,C 180,E1 -34029.519,E2 -34029.519} C_VEL
LIN {X 0,Y 42.356,Z 564.626,A -85,B 0,C 180,E1 -34020,E2 -34020} C_VEL
LIN {X 0,Y 46.879,Z 567.674,A -85,B 0,C 180,E1 -33993.369,E2 -33993.369} C_VEL
LIN {X 0,Y 49.959,Z 568.963,A -85,B 0,C 180,E1 -33985.887,E2 -33985.887} C_VEL
LIN {X 0,Y 39.875,Z 575.876,A -85,B 0,C 180,E1 -33977.825,E2 -33977.825} C_VEL
LIN {X 0,Y 35.457,Z 578.501,A -85,B 0,C 180,E1 -33973.352,E2 -33973.352} C_VEL
LIN {X 0,Y 27.348,Z 582.104,A -85,B 0,C 180,E1 -33965.143,E2 -33965.143} C_VEL
LIN {X 0,Y 21.238,Z 584.524,A -85,B 0,C 180,E1 -33954.245,E2 -33954.245} C_VEL
LIN {X 0,Y 18.033,Z 586.231,A -85,B 0,C 180,E1 -33940.307,E2 -33940.307} C_VEL
LIN {X 0,Y 17.477,Z 586.763,A -85,B 0,C 180,E1 -33934.4,E2 -33934.4} C_VEL
LIN {X 0,Y 17.705,Z 588.965,A -85,B 0,C 180,E1 -33906.755,E2 -33906.755} C_VEL
LIN {X 0,Y 25.521,Z 591.595,A -85,B 0,C 180,E1 -33874.646,E2 -33874.646} C_VEL
LIN {X 0,Y 37.253,Z 592.914,A -85,B 0,C 180,E1 -33860.01,E2 -33860.01} C_VEL
LIN {X 0,Y 50.247,Z 592.959,A -85,B 0,C 180,E1 -33852.724,E2 -33852.724} C_VEL
LIN {X 0,Y 63.725,Z 591.731,A -85,B 0,C 180,E1 -33848.519,E2 -33848.519} C_VEL
LIN {X 0,Y 77.448,Z 589.217,A -85,B 0,C 180,E1 -33845.951,E2 -33845.951} C_VEL
LIN {X 0,Y 91.286,Z 585.343,A -85,B 0,C 180,E1 -33844.211,E2 -33844.211} C_VEL
LIN {X 0,Y 91.238,Z 585.324,A -85,B 0,C 180,E1 -33843.779,E2 -33843.779} C_VEL
LIN {X 0,Y 77.062,Z 589.002,A -85,B 0,C 180,E1 -33841.637,E2 -33841.637} C_VEL
LIN {X 0,Y 63.043,Z 591.217,A -85,B 0,C 180,E1 -33838.515,E2 -33838.515} C_VEL
LIN {X 0,Y 49.308,Z 592.039,A -85,B 0,C 180,E1 -33833.734,E2 -33833.734} C_VEL
LIN {X 0,Y 36.138,Z 591.492,A -85,B 0,C 180,E1 -33825.612,E2 -33825.612} C_VEL
LIN {X 0,Y 24.348,Z 589.583,A -85,B 0,C 180,E1 -33809.58,E2 -33809.58} C_VEL
LIN {X 0,Y 19.799,Z 588.101,A -85,B 0,C 180,E1 -33794.965,E2 -33794.965} C_VEL
LIN {X 0,Y 16.818,Z 584.06,A -85,B 0,C 180,E1 -33749.942,E2 -33749.942} C_VEL
LIN {X 0,Y 21.414,Z 580,A -85,B 0,C 180,E1 -33720.566,E2 -33720.566} C_VEL
LIN {X 0,Y 29.164,Z 575.01,A -85,B 0,C 180,E1 -33703.855,E2 -33703.855} C_VEL
LIN {X 0,Y 38.343,Z 568.795,A -85,B 0,C 180,E1 -33693.656,E2 -33693.656} C_VEL
LIN {X 0,Y 41.137,Z 566.798,A -85,B 0,C 180,E1 -33691.598,E2 -33691.598} C_VEL
LIN {X 0,Y 41.871,Z 566.102,A -85,B 0,C 180,E1 -33690.123,E2 -33690.123} C_VEL
LIN {X 0,Y 36.578,Z 568.094,A -85,B 0,C 180,E1 -33671.039,E2 -33671.039} C_VEL
LIN {X 0,Y 36.448,Z 568.616,A -85,B 0,C 180,E1 -33660,E2 -33660} C_VEL
LIN {X 0,Y 38.654,Z 570.61,A -85,B 0,C 180,E1 -33638.751,E2 -33638.751} C_VEL
LIN {X 0,Y 40.457,Z 571.998,A -85,B 0,C 180,E1 -33630.005,E2 -33630.005} C_VEL
LIN {X 0,Y 31.295,Z 577.67,A -85,B 0,C 180,E1 -33621.62,E2 -33621.62} C_VEL
LIN {X 0,Y 21.339,Z 583.742,A -85,B 0,C 180,E1 -33599.549,E2 -33599.549} C_VEL
LIN {X 0,Y 17.477,Z 586.763,A -85,B 0,C 180,E1 -33574.4,E2 -33574.4} C_VEL
LIN {X 0,Y 16.571,Z 588.257,A -85,B 0,C 180,E1 -33555.293,E2 -33555.293} C_VEL
LIN {X 0,Y 17.726,Z 590.004,A -85,B 0,C 180,E1 -33522.459,E2 -33522.459} C_VEL
LIN {X 0,Y 21.971,Z 591.034,A -85,B 0,C 180,E1 -33503.067,E2 -33503.067} C_VEL
LIN {X 0,Y 26.727,Z 591.708,A -85,B 0,C 180,E1 -33494.88,E2 -33494.88} C_VEL
LIN {X 0,Y 28.527,Z 591.893,A -85,B 0,C 180,E1 -33493.264,E2 -33493.264} C_VEL
LIN {X 0,Y 42.281,Z 592.664,A -85,B 0,C 180,E1 -33486.507,E2 -33486.507} C_VEL
LIN {X 0,Y 49.171,Z 592.56,A -85,B 0,C 180,E1 -33484.588,E2 -33484.588} C_VEL
LIN {X 0,Y 52.746,Z 592.378,A -85,B 0,C 180,E1 -33483.186,E2 -33483.186} C_VEL
LIN {X 0,Y 41.71,Z 592.369,A -85,B 0,C 180,E1 -33480,E2 -33480} C_VEL
LIN {X 0,Y 28.201,Z 591.225,A -85,B 0,C 180,E1 -33473.151,E2 -33473.151} C_VEL
LIN {X 0,Y 14.626,Z 588.432,A -85,B 0,C 180,E1 -33451.387,E2 -33451.387} C_VEL
LIN {X 0,Y 9.625,Z 584.736,A -85,B 0,C 180,E1 -33389.898,E2 -33389.898} C_VEL
LIN {X 0,Y 15.575,Z 580.73,A -85,B 0,C 180,E1 -33347.495,E2 -33347.495} C_VEL
LIN {X 0,Y 24.754,Z 575.822,A -85,B 0,C 180,E1 -33331.838,E2 -33331.838} C_VEL
LIN {X 0,Y 31.815,Z 571.661,A -85,B 0,C 180,E1 -33325.944,E2 -33325.944} C_VEL
LIN {X 0,Y 32.256,Z 571.153,A -85,B 0,C 180,E1 -33322.116,E2 -33322.116} C_VEL
LIN {X 0,Y 30.656,Z 571.79,A -85,B 0,C 180,E1 -33313.208,E2 -33313.208} C_VEL
LIN {X 0,Y 30.378,Z 572.308,A -85,B 0,C 180,E1 -33300,E2 -33300} C_VEL
LIN {X 0,Y 32.038,Z 573.827,A -85,B 0,C 180,E1 -33279.52,E2 -33279.52} C_VEL
LIN {X 0,Y 30.74,Z 575.112,A -85,B 0,C 180,E1 -33275.779,E2 -33275.779} C_VEL
LIN {X 0,Y 21.234,Z 580.176,A -85,B 0,C 180,E1 -33265.637,E2 -33265.637} C_VEL
LIN {X 0,Y 13.124,Z 584.293,A -85,B 0,C 180,E1 -33242.343,E2 -33242.343} C_VEL
LIN {X 0,Y 11.533,Z 588.367,A -85,B 0,C 180,E1 -33172.711,E2 -33172.711} C_VEL
LIN {X 0,Y 22.264,Z 591.064,A -85,B 0,C 180,E1 -33139.429,E2 -33139.429} C_VEL
LIN {X 0,Y 28.527,Z 591.893,A -85,B 0,C 180,E1 -33133.264,E2 -33133.264} C_VEL
LIN {X 0,Y 28.174,Z 591.818,A -85,B 0,C 180,E1 -33131.511,E2 -33131.511} C_VEL
LIN {X 0,Y 26.622,Z 591.585,A -85,B 0,C 180,E1 -33129.669,E2 -33129.669} C_VEL
LIN {X 0,Y 20.704,Z 590.609,A -85,B 0,C 180,E1 -33125.901,E2 -33125.901} C_VEL
LIN {X 0,Y 9.335,Z 588.128,A -85,B 0,C 180,E1 -33116.854,E2 -33116.854} C_VEL
LIN {X 0,Y 3.299,Z 584.759,A -85,B 0,C 180,E1 -32996.429,E2 -32996.429} C_VEL
LIN {X 0,Y 14.851,Z 579.982,A -85,B 0,C 180,E1 -32959.193,E2 -32959.193} C_VEL
LIN {X 0,Y 23.504,Z 575.765,A -85,B 0,C 180,E1 -32955.083,E2 -32955.083} C_VEL
LIN {X 0,Y 24.217,Z 575.386,A -85,B 0,C 180,E1 -32950.542,E2 -32950.542} C_VEL
LIN {X 0,Y 24.204,Z 576.031,A -85,B 0,C 180,E1 -32933.928,E2 -32933.928} C_VEL
LIN {X 0,Y 23.57,Z 576.882,A -85,B 0,C 180,E1 -32927.15,E2 -32927.15} C_VEL
LIN {X 0,Y 11.424,Z 582.332,A -85,B 0,C 180,E1 -32917.104,E2 -32917.104} C_VEL
LIN {X 0,Y 3.024,Z 585.875,A -85,B 0,C 180,E1 -32850.323,E2 -32850.323} C_VEL
LIN {X 0,Y 14.042,Z 589.319,A -85,B 0,C 180,E1 -32764.839,E2 -32764.839} C_VEL
LIN {X 0,Y 14.003,Z 589.269,A -85,B 0,C 180,E1 -32762.268,E2 -32762.268} C_VEL
LIN {X 0,Y 2.404,Z 585.391,A -85,B 0,C 180,E1 -32669.593,E2 -32669.593} C_VEL
LIN {X 0,Y 3.299,Z 584.759,A -85,B 0,C 180,E1 -32636.429,E2 -32636.429} C_VEL
LIN {X 0,Y 5.489,Z 586.651,A -85,B 0,C 180,E1 -32616.247,E2 -32616.247} C_VEL
LIN {X 0,Y 5.489,Z 600,A -85,B 0,C 180,E1 -32616.247,E2 -32616.247} C_VEL
LIN {X 0,Y 5.489,Z 600,A -85,B 0,C 180,E1 -32616.247,E2 -32616.247}

QRS_NEXT_CUT()

QRS_NEXT()
QRS_HOME()

END
